// TwinCAT 3 PLC project PlcAly
// ProgramVersion: 3.1.4024.0
// libraries:
//   Tc2_EtherCAT, * (Beckhoff Automation GmbH)
//   Tc2_Standard, * (Beckhoff Automation GmbH)
//   Tc2_System, * (Beckhoff Automation GmbH)
//   Tc2_Utilities, * (Beckhoff Automation GmbH)
//   Tc3_Analytics, * (Beckhoff Automation GmbH)
//   Tc3_EventLogger, * (Beckhoff Automation GmbH)
//   Tc3_Module, * (Beckhoff Automation GmbH)
// project tree:
//   / AnalyticsTask.TcTTO, AnalyticsTask_C1.TcTTO, PlcTask.TcTTO
//   DUTs/Analytics/ E_AnalysisComponents.TcDUT, E_DataSourceContext.TcDUT, E_DataSourceState.TcDUT, E_DTType.TcDUT, E_ScopeCommand.TcDUT, E_VirtualInput.TcDUT, ST_AnalysisReset.TcDUT
//   DUTs/Analytics/HMI/Controls/ ST_HMI_C1_Ctrl1_Overall_Equipment_Effectiveness_OEE.TcDUT, ST_HMI_C1_Ctrl2_Machine_Learning_Calculation_Duration.TcDUT, ST_HMI_C1_Ctrl3_State_Unit.TcDUT
//   DUTs/Analytics/HMI/DataSourcePage/ E_SourceType.TcDUT, ST_HMI_DataSourceConfig.TcDUT, ST_HMI_DataSourceCtrl.TcDUT, ST_HMI_DataSourceHist.TcDUT, ST_HMI_DataSourceHistInfo.TcDUT, ST_HMI_DataSourceHistRecordInfo.TcDUT, ST_HMI_InputSource.TcDUT, ST_HMI_InputSourceCtrl.TcDUT
//   DUTs/Analytics/HMI/ ST_HMI_C1_OEE_Dashboard.TcDUT, ST_HMI_MapItem.TcDUT, ST_KeyValuePair.TcDUT
//   DUTs/Analytics/Sources/ ST_T1_Inputs.TcDUT
//   GVLs/ Analytics.TcGVL, AnalyticsHMI.TcGVL
//   POUs/Analytics/Analysis/ FB_Analysis.TcPOU
//   POUs/Analytics/Analysis/Networks/N01 OEEDashboard/ FB_N1_OEEDashboard.TcPOU
//   POUs/Analytics/Analysis/Networks/N01 OEEDashboard/Modules/ FB_N1_M1_State_Unit.TcPOU, FB_N1_M2_State_Execute.TcPOU, FB_N1_M3_State_Aborted.TcPOU, FB_N1_M4_State_Stopped.TcPOU, FB_N1_M5_Time_Scheduled.TcPOU, FB_N1_M6_OverallEquipmentEffectivenessOEE.TcPOU, FB_N1_M7_MachineLearningCalculationDuration.TcPOU
//   POUs/Analytics/Analysis/Networks/N01 OEEDashboard/N02 Products_Produced/ FB_N2_Products_Produced.TcPOU
//   POUs/Analytics/Analysis/Networks/N01 OEEDashboard/N02 Products_Produced/Modules/ FB_N2_M1_BatchNShift1Ch.TcPOU, FB_N2_M2_MathOperation.TcPOU, FB_N2_M3_EdgeCounter1Ch.TcPOU
//   POUs/Analytics/Analysis/Networks/N01 OEEDashboard/N03 Products_Defective/ FB_N3_Products_Defective.TcPOU
//   POUs/Analytics/Analysis/Networks/N01 OEEDashboard/N03 Products_Defective/Modules/ FB_N3_M1_BatchNShift1Ch.TcPOU, FB_N3_M2_MathOperation.TcPOU, FB_N3_M3_EdgeCounter1Ch.TcPOU
//   POUs/Analytics/Lambda/ FB_L1_Lf_CppModuleAssignString.TcPOU
//   POUs/Analytics/ MAIN_Analytics.TcPOU, MAIN_Analytics_C1.TcPOU
//   POUs/Analytics/Sources/T1_InputSource/ FB_T1_InputSource.TcPOU
//   POUs/Analytics/Sources/[Interfaces]/ I_InputSource.TcIO, I_InputSourceHistorical.TcIO
//   POUs/Analytics/VirtualInputSources/C1_AlyConfig/ FB_V1_C1_Virtual_Input_Source.TcPOU
//   POUs/Analytics/VirtualInputSources/[Interfaces]/ I_V1_Virtual_Input_Source.TcIO, I_VirtualInputSource.TcIO
//   POUs/Analytics/[Helper]/ FB_DataBuffer.TcPOU, FB_GetSampleIndex.TcPOU, FB_TcMessageSuccess.TcPOU, F_AlyTimestampToDCTimestruct.TcPOU, F_AlyTimestampToFileTime.TcPOU, F_AlyTimestampToLocalTime.TcPOU, F_ANY_Negation.TcPOU, F_ARRAY_To_LREAL_ARRAY.TcPOU, F_DCTimestructToFileTime.TcPOU, F_FileTimeToDCTimestruct.TcPOU, F_HasContext.TcPOU, F_SampleTimeCheck.TcPOU, F_ToANY.TcPOU
//   POUs/ MAIN.TcPOU
// (motion and I/O tree: see PLC project plc)
// real-time tasks:
//   TASK Task_Plc: cycle T#1ms, priority 5, ADS port 350
//   TASK Task_XPlanar_Hardware: cycle T#250us, priority 1, ADS port 351
//   TASK Task_XPlanar_Execute: cycle T#1ms, priority 3, ADS port 352
//   TASK Task_XPlanar_Prepare: cycle T#10ms, priority 10, ADS port 353
//   TASK Task_Job: cycle default, priority 7
//   TASK Task_Vision_Acquisition: cycle T#1ms, priority 4, ADS port 354
//   TASK Task_Vision_Display: cycle T#10ms, priority 12, ADS port 355
//   TASK Task_Vision_Execute: cycle T#10ms, priority 11, ADS port 356
//   TASK Task_IO: cycle T#50000us, priority 14, ADS port 301
//   TASK PlcTask: cycle T#10ms, priority 20, ADS port 357
//   TASK AnalyticsTask: cycle T#10ms, priority 21, ADS port 358
//   TASK AnalyticsTask_C1: cycle T#10ms, priority 22, ADS port 359
// variable links:

CONFIGURATION PlcAly
    RESOURCE PLC ON TwinCAT3
        TASK AnalyticsTask(INTERVAL := T#10ms, PRIORITY := 21);
        TASK AnalyticsTask_C1(INTERVAL := T#10ms, PRIORITY := 22);
        TASK PlcTask(INTERVAL := T#10ms, PRIORITY := 20);
        PROGRAM MAIN_Analytics WITH AnalyticsTask : MAIN_Analytics;
        PROGRAM MAIN_Analytics_C1 WITH AnalyticsTask_C1 : MAIN_Analytics_C1;
        PROGRAM MAIN WITH PlcTask : MAIN;
    END_RESOURCE
END_CONFIGURATION

// ---- DUTs/Analytics/E_AnalysisComponents.TcDUT
{attribute 'qualified_only'}
{attribute 'strict'}
TYPE E_AnalysisComponents : 
(
	All := -1,
	N1_OEEDashboard := 0,
	N1_M1_State_Unit := 1,
	N1_M2_State_Execute := 2,
	N1_M3_State_Aborted := 3,
	N1_M4_State_Stopped := 4,
	N1_M5_Time_Scheduled := 5,
	N1_M6_OverallEquipmentEffectivenessOEE := 6,
	N1_M7_MachineLearningCalculationDuration := 7,
	N2_Products_Produced := 8,
	N2_M1_BatchNShift1Ch := 9,
	N2_M2_MathOperation := 10,
	N2_M3_EdgeCounter1Ch := 11,
	N3_Products_Defective := 12,
	N3_M1_BatchNShift1Ch := 13,
	N3_M2_MathOperation := 14,
	N3_M3_EdgeCounter1Ch := 15,
	V1_Virtual_Input_Source := 16
) ;
END_TYPE

// ---- DUTs/Analytics/E_DataSourceContext.TcDUT
{attribute 'qualified_only'}
TYPE E_DataSourceContext : 
(
	eContext_No := 0, 
	eContext_Unknown := 2#0000_0000_0000_0001, //Unknown - All contexts allowed
	eContext_1000 := 2#0000_0000_0000_0010, //1000 µs
	eContext_Reserve1 := 2#0000_0000_0000_0100, //Reserve
	eContext_Reserve2 := 2#0000_0000_0000_1000, //Reserve
	eContext_Reserve3 := 2#0000_0000_0001_0000, //Reserve
	eContext_Reserve4 := 2#0000_0000_0010_0000, //Reserve
	eContext_Reserve5 := 2#0000_0000_0100_0000, //Reserve
	eContext_Reserve6 := 2#0000_0000_1000_0000, //Reserve
	eContext_Reserve7 := 2#0000_0001_0000_0000, //Reserve
	eContext_Reserve8 := 2#0000_0010_0000_0000, //Reserve
	eContext_Reserve9 := 2#0000_0100_0000_0000, //Reserve
	eContext_Reserve10 := 2#0000_1000_0000_0000, //Reserve
	eContext_Reserve11 := 2#0001_0000_0000_0000, //Reserve
	eContext_Reserve12 := 2#0010_0000_0000_0000, //Reserve
	eContext_Reserve13 := 2#0100_0000_0000_0000, //Reserve
	eContext_Reserve14 := 2#1000_0000_0000_0000 //Reserve
) DWORD;
END_TYPE

// ---- DUTs/Analytics/E_DataSourceState.TcDUT
{attribute 'qualified_only'}
{attribute 'strict'}
TYPE E_DataSourceState : 
(
	eUnknown := 0,
	eNotConnected,
	eReceiveData,
	eReceiveData_Cancel,
	eReceiveData_Pause,
	eError,
	eReady,
	eWaitForData
) ;
END_TYPE

// ---- DUTs/Analytics/E_DTType.TcDUT
{attribute 'qualified_only'}
{attribute 'strict'}
TYPE E_DTType : 
(
	NotInitialized := 0,
	BOOL_,
	BYTE_,
	WORD_,
	DWORD_,
	SINT_,
	USINT_,
	INT_,
	UINT_,
	DINT_,
	UDINT_,
	LINT_,
	ULINT_,
	REAL_,
	LREAL_,
	LWORD_
) ;
END_TYPE

// ---- DUTs/Analytics/E_ScopeCommand.TcDUT
{attribute 'qualified_only'}
{attribute 'strict'}
TYPE E_ScopeCommand : 
(
	eDefault := 0,
	ePause,
	eStop
) ;
END_TYPE

// ---- DUTs/Analytics/E_VirtualInput.TcDUT
{attribute 'qualified_only'}
TYPE E_VirtualInput : 
(
	eContext_No := 0, 
	eContext_V1_Virtual_Input_Source := 2#0000_0000_0000_0001_0000_0000_0000_0000, //Virtual_Input_Source
	eContext_Vn_Reserve1 := 2#0000_0000_0000_0010_0000_0000_0000_0000, //Reserve
	eContext_Vn_Reserve2 := 2#0000_0000_0000_0100_0000_0000_0000_0000, //Reserve
	eContext_Vn_Reserve3 := 2#0000_0000_0000_1000_0000_0000_0000_0000, //Reserve
	eContext_Vn_Reserve4 := 2#0000_0000_0001_0000_0000_0000_0000_0000, //Reserve
	eContext_Vn_Reserve5 := 2#0000_0000_0010_0000_0000_0000_0000_0000, //Reserve
	eContext_Vn_Reserve6 := 2#0000_0000_0100_0000_0000_0000_0000_0000, //Reserve
	eContext_Vn_Reserve7 := 2#0000_0000_1000_0000_0000_0000_0000_0000, //Reserve
	eContext_Vn_Reserve8 := 2#0000_0001_0000_0000_0000_0000_0000_0000, //Reserve
	eContext_Vn_Reserve9 := 2#0000_0010_0000_0000_0000_0000_0000_0000, //Reserve
	eContext_Vn_Reserve10 := 2#0000_0100_0000_0000_0000_0000_0000_0000, //Reserve
	eContext_Vn_Reserve11 := 2#0000_1000_0000_0000_0000_0000_0000_0000, //Reserve
	eContext_Vn_Reserve12 := 2#0001_0000_0000_0000_0000_0000_0000_0000, //Reserve
	eContext_Vn_Reserve13 := 2#0010_0000_0000_0000_0000_0000_0000_0000, //Reserve
	eContext_Vn_Reserve14 := 2#0100_0000_0000_0000_0000_0000_0000_0000, //Reserve
	eContext_Vn_Reserve15 := 2#1000_0000_0000_0000_0000_0000_0000_0000 //Reserve
) DWORD;
END_TYPE

// ---- DUTs/Analytics/HMI/Controls/ST_HMI_C1_Ctrl1_Overall_Equipment_Effectiveness_OEE.TcDUT
TYPE ST_HMI_C1_Ctrl1_Overall_Equipment_Effectiveness_OEE : 
STRUCT
	//Overall Equipment Effectiveness (OEE)
	bTrigReconfigure: BOOL;
	fM6_fOEE: LREAL; //Overall equipment effectiveness (OEE)
	fM6_fAvailability: LREAL; //Availability
	fM6_fPerformance: LREAL; //Performance
	fM6_fQuality: LREAL; //Quality
	fM6_fThresholdLevelOkWarning: LREAL; //Level Ok / Warning
	fM6_fThresholdLevelWarningAlarm: LREAL; //Level Warning / Alarm
	eM6_eOeeClass: E_ALY_Classification_3Cls; //OEE Classification
END_STRUCT
END_TYPE

// ---- DUTs/Analytics/HMI/Controls/ST_HMI_C1_Ctrl2_Machine_Learning_Calculation_Duration.TcDUT
TYPE ST_HMI_C1_Ctrl2_Machine_Learning_Calculation_Duration : 
STRUCT
	//Machine Learning Calculation Duration
	bTrigReconfigure: BOOL;
	nM7_nDataIn: UDINT; //Actual Value
	fM7_fMin: LREAL; //Min Value
	fM7_fMax: LREAL; //Max Value
	fM7_fAvg: LREAL; //Avg Value
	tM7_fbTimeMin: DCTIMESTRUCT; //Last Event Min
	tM7_fbTimeMax: DCTIMESTRUCT; //Last Event Max
END_STRUCT
END_TYPE

// ---- DUTs/Analytics/HMI/Controls/ST_HMI_C1_Ctrl3_State_Unit.TcDUT
TYPE ST_HMI_C1_Ctrl3_State_Unit : 
STRUCT
	//State_Unit
	bTrigReconfigure: BOOL;
	sM1_sOutput: STRING(255); //Value
END_STRUCT
END_TYPE

// ---- DUTs/Analytics/HMI/DataSourcePage/E_SourceType.TcDUT
{attribute 'qualified_only'}
{attribute 'strict'}
TYPE E_SourceType : 
(
	eLive := 0,
	eHistMQTT,
	eHistFile
) ;
END_TYPE

// ---- DUTs/Analytics/HMI/DataSourcePage/ST_HMI_DataSourceConfig.TcDUT
TYPE ST_HMI_DataSourceConfig : 
STRUCT
	nID: DINT;
	sDisplayName: WSTRING(80);
	eConfigType: E_SourceType;
	aInputSources: ARRAY [0..0] OF ST_HMI_InputSource;
END_STRUCT
END_TYPE

// ---- DUTs/Analytics/HMI/DataSourcePage/ST_HMI_DataSourceCtrl.TcDUT
TYPE ST_HMI_DataSourceCtrl : 
STRUCT
	nActiveConfigurationIdx: INT;
	
	aInputSourceCtrls: ARRAY [0..0] OF ST_HMI_InputSourceCtrl;
	
	bStart: BOOL;
	bCancel: BOOL;
	bPause: BOOL;
	bReset: BOOL;
	
	bUpdateRecordList: BOOL;
END_STRUCT
END_TYPE

// ---- DUTs/Analytics/HMI/DataSourcePage/ST_HMI_DataSourceHist.TcDUT
TYPE ST_HMI_DataSourceHist : 
STRUCT
	nCurrentRecordID: DINT;
	stSourceInfo: ST_HMI_DataSourceHistInfo;
	nRecordCount: DINT;
	aRecords: ARRAY [0..255] OF ST_HMI_DataSourceHistRecordInfo;
END_STRUCT
END_TYPE

// ---- DUTs/Analytics/HMI/DataSourcePage/ST_HMI_DataSourceHistInfo.TcDUT
TYPE ST_HMI_DataSourceHistInfo : 
STRUCT
	sSPGuid: GUID;
	sAlyFilePath: STRING(255);
	sSourceType: STRING(80);
	sTopic: STRING(255);
	sLayoutID: GUID;
	sAlias: STRING(255);
END_STRUCT
END_TYPE

// ---- DUTs/Analytics/HMI/DataSourcePage/ST_HMI_DataSourceHistRecordInfo.TcDUT
TYPE ST_HMI_DataSourceHistRecordInfo : 
STRUCT
	nID: DINT;
	sName: WSTRING(80);
	sDisplayName: WSTRING(80);
	dtRecordStart: DCTIMESTRUCT;
	dtRecordEnd: DCTIMESTRUCT;
	dtSelectedRangeStart: DCTIMESTRUCT;
	dtSelectedRangeEnd: DCTIMESTRUCT;
END_STRUCT
END_TYPE

// ---- DUTs/Analytics/HMI/DataSourcePage/ST_HMI_InputSource.TcDUT
TYPE ST_HMI_InputSource : 
STRUCT
	nID: DINT;
	sDisplayName: WSTRING(80);
	
	sStreamSystemID: GUID;
	sTopic: STRING(255);
	
	eSourceType: E_SourceType;;
	eState: E_DataSourceState;;
	dtTimestamp: DCTIMESTRUCT;
	
	stHist: ST_HMI_DataSourceHist;
END_STRUCT
END_TYPE

// ---- DUTs/Analytics/HMI/DataSourcePage/ST_HMI_InputSourceCtrl.TcDUT
TYPE ST_HMI_InputSourceCtrl : 
STRUCT
	nActiveRecordIdx: INT;
	
	dtSelectedRangeStart: DCTIMESTRUCT;
	dtSelectedRangeEnd: DCTIMESTRUCT;
	
	bStart: BOOL;
	bCancel: BOOL;
	bPause: BOOL;
	bReset: BOOL;
END_STRUCT
END_TYPE

// ---- DUTs/Analytics/HMI/ST_HMI_C1_OEE_Dashboard.TcDUT
TYPE ST_HMI_C1_OEE_Dashboard : 
STRUCT
	stHMI_C1_Ctrl3_State_Unit: ST_HMI_C1_Ctrl3_State_Unit;
	
	stHMI_C1_Ctrl1_Overall_Equipment_Effectiveness_OEE: ST_HMI_C1_Ctrl1_Overall_Equipment_Effectiveness_OEE;
	
	stHMI_C1_Ctrl2_Machine_Learning_Calculation_Duration: ST_HMI_C1_Ctrl2_Machine_Learning_Calculation_Duration;
END_STRUCT
END_TYPE

// ---- DUTs/Analytics/HMI/ST_HMI_MapItem.TcDUT
TYPE ST_HMI_MapItem : 
STRUCT
	sName: WSTRING(127);
	sDescription: WSTRING(127);
	sPosition: WSTRING(127);
	nStatus: INT;
END_STRUCT
END_TYPE

// ---- DUTs/Analytics/HMI/ST_KeyValuePair.TcDUT
TYPE ST_KeyValuePair : 
STRUCT
	sKey: WSTRING(127);
	sValue: STRING(255);
END_STRUCT
END_TYPE

// ---- DUTs/Analytics/Sources/ST_T1_Inputs.TcDUT
TYPE ST_T1_Inputs : 
STRUCT
	nGVL_Components_fbMachine_stAnalytics_nState: UINT; //GVL_Components.fbMachine.stAnalytics.nState
	nGVL_Components_fbMachine_stAnalytics_nUnitsProduced: ULINT; //GVL_Components.fbMachine.stAnalytics.nUnitsProduced
	nGVL_Components_fbMachine_stAnalytics_nDefectiveUnits: ULINT; //GVL_Components.fbMachine.stAnalytics.nDefectiveUnits
	nGVL_Components_fbMachine_stAnalytics_tMlCalculation: UDINT; //GVL_Components.fbMachine.stAnalytics.tMlCalculation
END_STRUCT
END_TYPE

// ---- DUTs/Analytics/ST_AnalysisReset.TcDUT
TYPE ST_AnalysisReset : 
STRUCT
	eResetComponent: E_AnalysisComponents := E_AnalysisComponents.All;
	bResetExecute: BOOL;
END_STRUCT
END_TYPE

// ---- GVLs/Analytics.TcGVL
{attribute 'qualified_only'}
VAR_GLOBAL
	//DataSources
	//Live:
	fbT1_InputSource: FB_T1_InputSource;
	//Historical:
	//Empty:
	
	fbT1_IecCriticalSection: FB_IecCriticalSection;
	
	//Historical DataSource parameter
	nHistMaxInputBuffer: UDINT := 100;
	nHistMaxSampleCount: UDINT := 100;
	
	stReset: ST_AnalysisReset;
END_VAR

// ---- GVLs/AnalyticsHMI.TcGVL
{attribute 'qualified_only'}
VAR_GLOBAL
	//Switch between historical and live data
	stHMI_DataSourceCtrl: ST_HMI_DataSourceCtrl;
	stHMI_DataSourceConfig: ARRAY [0..0] OF ST_HMI_DataSourceConfig := [ 
																	( nID:= 1, sDisplayName:= "AlyConfig", eConfigType:= E_SourceType.eLive, 
																		aInputSources:= [ 
																			( nID:= 1, sDisplayName:= "00436273-58a1-a0ec-e33c-07029f4f38f0", sStreamSystemID:= STRING_TO_GUID('00436273-58a1-a0ec-e33c-07029f4f38f0'), 
																				sTopic:= 'DefaultMainTopic/PlcStream1', eSourceType:= E_SourceType.eLive, eState:= E_DataSourceState.eUnknown ) ] ) ];
	
	//Reset
	bN1_OEEDashboard_Reset: BOOL;
	bN1_M1_State_Unit_Reset: BOOL;
	bN1_M2_State_Execute_Reset: BOOL;
	bN1_M3_State_Aborted_Reset: BOOL;
	bN1_M4_State_Stopped_Reset: BOOL;
	bN1_M5_Time_Scheduled_Reset: BOOL;
	bN1_M6_OverallEquipmentEffectivenessOEE_Reset: BOOL;
	bN1_M7_MachineLearningCalculationDuration_Reset: BOOL;
	bN2_Products_Produced_Reset: BOOL;
	bN2_M1_BatchNShift1Ch_Reset: BOOL;
	bN2_M2_MathOperation_Reset: BOOL;
	bN2_M3_EdgeCounter1Ch_Reset: BOOL;
	bN3_Products_Defective_Reset: BOOL;
	bN3_M1_BatchNShift1Ch_Reset: BOOL;
	bN3_M2_MathOperation_Reset: BOOL;
	bN3_M3_EdgeCounter1Ch_Reset: BOOL;
	
	//HMI Structs
	stHMI_C1_OEE_Dashboard: ST_HMI_C1_OEE_Dashboard;
	
	//HMI Map Items
	aMapItems: ARRAY [0..0] OF ST_HMI_MapItem := [(sName:="00436273-58a1-a0ec-e33c-07029f4f38f0", sDescription:="", sPosition:="", nStatus:= 0)];
END_VAR

// ---- POUs/Analytics/Sources/[Interfaces]/I_InputSource.TcIO
INTERFACE I_InputSource

METHOD AddClient : BOOL
VAR_OUTPUT
	nClientID: LWORD;
END_VAR
END_METHOD

METHOD Call : BOOL
END_METHOD

METHOD ClientDone : BOOL
VAR_INPUT
	nClientID: LWORD;
END_VAR
END_METHOD

METHOD GetData : BOOL
VAR_INPUT
	nElement: UDINT;
	pInputs: PVOID;
	nInputsSize: UDINT;
END_VAR
VAR_OUTPUT
	nTimestamp: ULINT;
	nContext: DWORD;
END_VAR
END_METHOD

METHOD NewDataAvailable : BOOL
VAR_INPUT
	nLastDataHandle: ULINT;
END_VAR
END_METHOD

PROPERTY eDataState : E_DataSourceState
GET
END_GET
END_PROPERTY

PROPERTY bReadNewData : BOOL
GET
END_GET
END_PROPERTY

PROPERTY nDataHandle : ULINT
GET
END_GET
END_PROPERTY

PROPERTY nElements : UDINT
GET
END_GET
END_PROPERTY

PROPERTY nMaxOversamplingFactor : UDINT
GET
END_GET
END_PROPERTY

END_INTERFACE

// ---- POUs/Analytics/Sources/[Interfaces]/I_InputSourceHistorical.TcIO
INTERFACE I_InputSourceHistorical EXTENDS I_InputSource

METHOD HistoricalCtrl : BOOL
VAR_INPUT
	stCtrl: REFERENCE TO ST_HMI_InputSourceCtrl;
	stHistStreamInfo: REFERENCE TO ST_HMI_DataSourceHist;
	stRecordInfo: REFERENCE TO ST_HMI_DataSourceHistRecordInfo;
END_VAR
END_METHOD

METHOD UpdateRecordList : BOOL
VAR_INPUT
	sStreamSystemID: GUID;
	stHistStreamInfo: REFERENCE TO ST_HMI_DataSourceHist;
END_VAR
END_METHOD

PROPERTY bCtrlChanged : BOOL
GET
END_GET
END_PROPERTY

END_INTERFACE

// ---- POUs/Analytics/VirtualInputSources/[Interfaces]/I_V1_Virtual_Input_Source.TcIO
INTERFACE I_V1_Virtual_Input_Source EXTENDS I_VirtualInputSource

PROPERTY nV1_tMlCalculation : UDINT
GET
END_GET
END_PROPERTY

PROPERTY nV1_nUnitsProduced : ULINT
GET
END_GET
END_PROPERTY

PROPERTY nV1_nDefectiveUnits : ULINT
GET
END_GET
END_PROPERTY

PROPERTY nV1_nState : UINT
GET
END_GET
END_PROPERTY

END_INTERFACE

// ---- POUs/Analytics/VirtualInputSources/[Interfaces]/I_VirtualInputSource.TcIO
INTERFACE I_VirtualInputSource

METHOD Done : BOOL
END_METHOD

METHOD NextData : BOOL
VAR_INPUT
	nMaxOversampling: UDINT;
END_VAR
END_METHOD

METHOD SourceSync : BOOL
END_METHOD

PROPERTY bEndOfData : BOOL
GET
END_GET
END_PROPERTY

PROPERTY dtTimestamp : DCTIMESTRUCT
GET
END_GET
END_PROPERTY

PROPERTY nContext : DWORD
GET
END_GET
END_PROPERTY

PROPERTY nDataHandle : ULINT
GET
END_GET
END_PROPERTY

PROPERTY tTimestamp : ULINT
GET
END_GET
END_PROPERTY

PROPERTY eSourceState : E_DataSourceState
GET
END_GET
END_PROPERTY

END_INTERFACE

// ---- POUs/Analytics/MAIN_Analytics.TcPOU
PROGRAM MAIN_Analytics
VAR
END_VAR


//Reset Analytics Components
A_Reset();

CASE AnalyticsHMI.stHMI_DataSourceCtrl.nActiveConfigurationIdx OF
	0:

		//Reset
		MAIN_Analytics_C1.A_Reset(stReset := Analytics.stReset);

		//Map to HMI
		MAIN_Analytics_C1.A_MapToHMI();
END_CASE


//Call DataSource FBs
IF Analytics.fbT1_InputSource.bReadNewData THEN
	Analytics.fbT1_InputSource.Call();
END_IF

ACTION A_Reset:

IF AnalyticsHMI.bN1_OEEDashboard_Reset THEN
	Analytics.stReset.eResetComponent:= E_AnalysisComponents.N1_OEEDashboard;
	Analytics.stReset.bResetExecute:= TRUE;
	AnalyticsHMI.bN1_OEEDashboard_Reset:= FALSE;
END_IF

IF AnalyticsHMI.bN1_M1_State_Unit_Reset THEN
	Analytics.stReset.eResetComponent:= E_AnalysisComponents.N1_M1_State_Unit;
	Analytics.stReset.bResetExecute:= TRUE;
	AnalyticsHMI.bN1_M1_State_Unit_Reset:= FALSE;
END_IF

IF AnalyticsHMI.bN1_M2_State_Execute_Reset THEN
	Analytics.stReset.eResetComponent:= E_AnalysisComponents.N1_M2_State_Execute;
	Analytics.stReset.bResetExecute:= TRUE;
	AnalyticsHMI.bN1_M2_State_Execute_Reset:= FALSE;
END_IF

IF AnalyticsHMI.bN1_M3_State_Aborted_Reset THEN
	Analytics.stReset.eResetComponent:= E_AnalysisComponents.N1_M3_State_Aborted;
	Analytics.stReset.bResetExecute:= TRUE;
	AnalyticsHMI.bN1_M3_State_Aborted_Reset:= FALSE;
END_IF

IF AnalyticsHMI.bN1_M4_State_Stopped_Reset THEN
	Analytics.stReset.eResetComponent:= E_AnalysisComponents.N1_M4_State_Stopped;
	Analytics.stReset.bResetExecute:= TRUE;
	AnalyticsHMI.bN1_M4_State_Stopped_Reset:= FALSE;
END_IF

IF AnalyticsHMI.bN1_M5_Time_Scheduled_Reset THEN
	Analytics.stReset.eResetComponent:= E_AnalysisComponents.N1_M5_Time_Scheduled;
	Analytics.stReset.bResetExecute:= TRUE;
	AnalyticsHMI.bN1_M5_Time_Scheduled_Reset:= FALSE;
END_IF

IF AnalyticsHMI.bN1_M6_OverallEquipmentEffectivenessOEE_Reset THEN
	Analytics.stReset.eResetComponent:= E_AnalysisComponents.N1_M6_OverallEquipmentEffectivenessOEE;
	Analytics.stReset.bResetExecute:= TRUE;
	AnalyticsHMI.bN1_M6_OverallEquipmentEffectivenessOEE_Reset:= FALSE;
END_IF

IF AnalyticsHMI.bN1_M7_MachineLearningCalculationDuration_Reset THEN
	Analytics.stReset.eResetComponent:= E_AnalysisComponents.N1_M7_MachineLearningCalculationDuration;
	Analytics.stReset.bResetExecute:= TRUE;
	AnalyticsHMI.bN1_M7_MachineLearningCalculationDuration_Reset:= FALSE;
END_IF

IF AnalyticsHMI.bN2_Products_Produced_Reset THEN
	Analytics.stReset.eResetComponent:= E_AnalysisComponents.N2_Products_Produced;
	Analytics.stReset.bResetExecute:= TRUE;
	AnalyticsHMI.bN2_Products_Produced_Reset:= FALSE;
END_IF

IF AnalyticsHMI.bN2_M1_BatchNShift1Ch_Reset THEN
	Analytics.stReset.eResetComponent:= E_AnalysisComponents.N2_M1_BatchNShift1Ch;
	Analytics.stReset.bResetExecute:= TRUE;
	AnalyticsHMI.bN2_M1_BatchNShift1Ch_Reset:= FALSE;
END_IF

IF AnalyticsHMI.bN2_M2_MathOperation_Reset THEN
	Analytics.stReset.eResetComponent:= E_AnalysisComponents.N2_M2_MathOperation;
	Analytics.stReset.bResetExecute:= TRUE;
	AnalyticsHMI.bN2_M2_MathOperation_Reset:= FALSE;
END_IF

IF AnalyticsHMI.bN2_M3_EdgeCounter1Ch_Reset THEN
	Analytics.stReset.eResetComponent:= E_AnalysisComponents.N2_M3_EdgeCounter1Ch;
	Analytics.stReset.bResetExecute:= TRUE;
	AnalyticsHMI.bN2_M3_EdgeCounter1Ch_Reset:= FALSE;
END_IF

IF AnalyticsHMI.bN3_Products_Defective_Reset THEN
	Analytics.stReset.eResetComponent:= E_AnalysisComponents.N3_Products_Defective;
	Analytics.stReset.bResetExecute:= TRUE;
	AnalyticsHMI.bN3_Products_Defective_Reset:= FALSE;
END_IF

IF AnalyticsHMI.bN3_M1_BatchNShift1Ch_Reset THEN
	Analytics.stReset.eResetComponent:= E_AnalysisComponents.N3_M1_BatchNShift1Ch;
	Analytics.stReset.bResetExecute:= TRUE;
	AnalyticsHMI.bN3_M1_BatchNShift1Ch_Reset:= FALSE;
END_IF

IF AnalyticsHMI.bN3_M2_MathOperation_Reset THEN
	Analytics.stReset.eResetComponent:= E_AnalysisComponents.N3_M2_MathOperation;
	Analytics.stReset.bResetExecute:= TRUE;
	AnalyticsHMI.bN3_M2_MathOperation_Reset:= FALSE;
END_IF

IF AnalyticsHMI.bN3_M3_EdgeCounter1Ch_Reset THEN
	Analytics.stReset.eResetComponent:= E_AnalysisComponents.N3_M3_EdgeCounter1Ch;
	Analytics.stReset.bResetExecute:= TRUE;
	AnalyticsHMI.bN3_M3_EdgeCounter1Ch_Reset:= FALSE;
END_IF
END_ACTION

END_PROGRAM

// ---- POUs/Analytics/MAIN_Analytics_C1.TcPOU
PROGRAM MAIN_Analytics_C1
VAR_INPUT
	stReset: ST_AnalysisReset;
END_VAR
VAR_OUTPUT
	bError: BOOL;
	ipTcResult: I_TcMessage;
END_VAR
VAR
	nHMIUpdateState: INT;
	bHMIReinit: BOOL := TRUE;
	bHMIResetReinit: BOOL;
	bHMIReinitDone: BOOL;
	
	fbV1_C1_Virtual_Input_Source: FB_V1_C1_Virtual_Input_Source(fbSource:= Analytics.fbT1_InputSource);
	
	fbAnalysis: FB_Analysis := ( nConfigurationID:= 1, 
								ipVirtual_Input_Source:= fbV1_C1_Virtual_Input_Source );
END_VAR

A_Reset();

fbV1_C1_Virtual_Input_Source.SourceSync();

IF NOT fbV1_C1_Virtual_Input_Source.bEndOfData THEN

	WHILE NOT fbV1_C1_Virtual_Input_Source.bEndOfData DO

		fbV1_C1_Virtual_Input_Source.NextData(1);

		fbAnalysis.Call();

	END_WHILE

ELSE
	fbAnalysis.Call();
END_IF

fbV1_C1_Virtual_Input_Source.Done();

//Error Handling
bError:= fbAnalysis.bError;
ipTcResult:= fbAnalysis.ipTcResult;


//Map HMI Current Timestamp
AnalyticsHMI.stHMI_DataSourceConfig[0].aInputSources[0].eState:= fbV1_C1_Virtual_Input_Source.fbInputSource.eDataState;
AnalyticsHMI.stHMI_DataSourceConfig[0].aInputSources[0].dtTimestamp:= fbV1_C1_Virtual_Input_Source.dtTimestamp;

ACTION A_Reset:

//Reset Analytics Components
fbAnalysis.Reset(stReset);

Analytics.stReset.bResetExecute:= FALSE;
END_ACTION

ACTION A_MapToHMI:

//Map In-/Outputs of the Analysis to HMI Structs
CASE nHMIUpdateState OF
	0:
		bHMIReinit:= bHMIReinit OR fbAnalysis.GetHMIValues(1, ADR(AnalyticsHMI.stHMI_C1_OEE_Dashboard));
		bHMIReinitDone:= fbAnalysis.SetHMIValues(1, ADR(AnalyticsHMI.stHMI_C1_OEE_Dashboard), bHMIReinit);
		nHMIUpdateState:= 1;
	1:
		IF bHMIResetReinit THEN
			bHMIResetReinit:= FALSE;
			bHMIReinit:= FALSE;
		END_IF

		IF bHMIReinitDone THEN
			bHMIResetReinit:= TRUE;
		END_IF

		nHMIUpdateState:= 0;
END_CASE
END_ACTION

END_PROGRAM

// ---- POUs/Analytics/VirtualInputSources/C1_AlyConfig/FB_V1_C1_Virtual_Input_Source.TcPOU
FUNCTION_BLOCK FB_V1_C1_Virtual_Input_Source IMPLEMENTS I_VirtualInputSource, I_V1_Virtual_Input_Source
VAR
	_fbSource: I_InputSource;
	
	_nSourceClientID: LWORD;
	_nDataHandle: ULINT;
	_nElements: UDINT;
	
	_nSelectedElement: UDINT;
	_nSelectedOversample: UDINT;
	
	_nContext: DWORD;
	_stInputs: ST_T1_Inputs;
	
	_nTimestamp: ULINT;
END_VAR

PROPERTY bEndOfData : BOOL
GET
bEndOfData:= _nElements = 0 OR (_nSelectedElement >= _nElements AND _nSelectedOversample >= _fbSource.nMaxOversamplingFactor);
END_GET
END_PROPERTY

METHOD Done : BOOL
VAR
END_VAR
IF bEndOfData AND _nElements > 0 THEN
	_nElements:= 0;
	_fbSource.ClientDone(_nSourceClientID);
END_IF

_nContext:= 0;
END_METHOD

PROPERTY dtTimestamp : DCTIMESTRUCT
GET
dtTimestamp:= F_AlyTimestampToDCTimestruct(_nTimestamp);
END_GET
END_PROPERTY

PROPERTY eSourceState : E_DataSourceState
GET
eSourceState:= _fbSource.eDataState;
END_GET
END_PROPERTY

METHOD FB_init : BOOL
VAR_INPUT
	bInitRetains: BOOL; // if TRUE, the retain variables are initialized (warm start / cold start)
	bInCopyCode: BOOL; // if TRUE, the instance afterwards gets moved into the copy code (online change)
	fbSource: I_InputSource;
END_VAR
VAR
END_VAR
IF NOT bInCopyCode THEN
	fbSource.AddClient(nClientID=>_nSourceClientID);
	_fbSource:= fbSource;
END_IF
END_METHOD

PROPERTY fbInputSource : I_InputSource
GET
fbInputSource:= _fbSource;
END_GET
END_PROPERTY

PROPERTY nContext : DWORD
GET
nContext:= _nContext;
END_GET
END_PROPERTY

PROPERTY nDataHandle : ULINT
GET
nDataHandle:= _nDataHandle;
END_GET
END_PROPERTY

METHOD NextData : BOOL
VAR_INPUT
	nMaxOversampling: UDINT;
END_VAR
VAR
END_VAR
IF _nElements > 0 AND NOT bEndOfData THEN

	_nSelectedOversample:= _nSelectedOversample + 1;
	IF _nSelectedOversample > nMaxOversampling OR _nSelectedElement = 0 THEN
		_nSelectedElement:= _nSelectedElement + 1;
		_nSelectedOversample:= 1;
	END_IF

	NextData:= _fbSource.GetData(_nSelectedElement, ADR(_stInputs), SIZEOF(_stInputs), nTimestamp=>_nTimestamp, nContext=>_nContext);
	_nContext:= _nContext OR E_VirtualInput.eContext_V1_Virtual_Input_Source;
END_IF
END_METHOD

PROPERTY nV1_nDefectiveUnits : ULINT
GET
nV1_nDefectiveUnits:= _stInputs.nGVL_Components_fbMachine_stAnalytics_nDefectiveUnits;
END_GET
END_PROPERTY

PROPERTY nV1_nState : UINT
GET
nV1_nState:= _stInputs.nGVL_Components_fbMachine_stAnalytics_nState;
END_GET
END_PROPERTY

PROPERTY nV1_nUnitsProduced : ULINT
GET
nV1_nUnitsProduced:= _stInputs.nGVL_Components_fbMachine_stAnalytics_nUnitsProduced;
END_GET
END_PROPERTY

PROPERTY nV1_tMlCalculation : UDINT
GET
nV1_tMlCalculation:= _stInputs.nGVL_Components_fbMachine_stAnalytics_tMlCalculation;
END_GET
END_PROPERTY

METHOD SourceSync : BOOL
VAR
END_VAR
IF _fbSource.NewDataAvailable(_nDataHandle) THEN
	_nDataHandle:= _fbSource.nDataHandle;
	_nElements:= _fbSource.nElements;

	_nSelectedElement:= 0;
	_nSelectedOversample:= 0;
END_IF
END_METHOD

PROPERTY tTimestamp : ULINT
GET
tTimestamp:= _nTimestamp;
END_GET
END_PROPERTY

END_FUNCTION_BLOCK

// ---- POUs/Analytics/[Helper]/F_AlyTimestampToDCTimestruct.TcPOU
FUNCTION F_AlyTimestampToDCTimestruct : DCTIMESTRUCT
VAR_INPUT
	tTimestamp: ULINT;
END_VAR
VAR
	tFileTime: T_FILETIME;
	newDCTime: T_DCTIME64;
	
	fbToLocal: FB_FileTimeToTzSpecificLocalTime;
	//W. Europe Daylight Time
	//(UTC+01:00) Amsterdam, Berlin, Bern, Rome, Stockholm, Vienna
	tzInfo: ST_TimeZoneInformation := (bias := -60, standardDate := (wMonth := 10 ,wDay:=5, wHour := 3), daylightDate := (wMonth := 3, wDay:=5, wHour := 2), daylightBias := -60);
END_VAR

tFileTime:= DCTIME64_TO_Filetime(tTimestamp);
fbToLocal(in:= tFileTime, tzInfo:= tzInfo);
newDCTime:= FILETIME_TO_DCTIME64(fbToLocal.out);

F_AlyTimestampToDCTimestruct:= DCTIME64_TO_DCTIMESTRUCT(newDCTime);

END_FUNCTION

// ---- POUs/Analytics/Analysis/FB_Analysis.TcPOU
FUNCTION_BLOCK FB_Analysis
VAR_INPUT
	nConfigurationID: INT;
	ipVirtual_Input_Source: I_V1_Virtual_Input_Source;
	
END_VAR
VAR_OUTPUT
	bError: BOOL;
	ipTcResult: I_TcMessage := fbTcMsgSuccess;
END_VAR
VAR
	fbTcMsgSuccess: FB_TcMessageSuccess;
	
	R_TRIG_Reset: R_TRIG;
	bResetBusy: BOOL;
	
	fbN1_OEEDashboard: FB_N1_OEEDashboard;
END_VAR

METHOD Call : BOOL
VAR
END_VAR

//Analytics Network "OEEDashboard" with ID: 1
fbN1_OEEDashboard.Call(THIS);


//Error Handling
IF fbN1_OEEDashboard.bError THEN
	bError:= TRUE;
	ipTcResult:= fbN1_OEEDashboard.ipTcResult;
ELSE
	bError:= FALSE;
	ipTcResult:= fbTcMsgSuccess;
END_IF
END_METHOD

METHOD GetHMIValues : BOOL
VAR_INPUT
	nContentID: DINT;
	pContent: PVOID;
END_VAR
VAR
END_VAR

CASE nContentID OF
	1:
		GetHMIValues:= GetHMIValues OR fbN1_OEEDashboard.fbM6_OverallEquipmentEffectivenessOEE.GetHMI(1, pContent);
END_CASE
END_METHOD

PROPERTY nContext : DWORD
GET

nContext:= 0;
IF ipVirtual_Input_Source <> 0 THEN
	nContext:= ipVirtual_Input_Source.nContext;
END_IF
END_GET
END_PROPERTY

METHOD Reset : BOOL
VAR_IN_OUT
	stReset: ST_AnalysisReset;
END_VAR
VAR
END_VAR

R_TRIG_Reset(CLK:= stReset.bResetExecute);
IF R_TRIG_Reset.Q OR bResetBusy THEN
	bResetBusy:= TRUE;

	CASE stReset.eResetComponent OF
		E_AnalysisComponents.All:
			bResetBusy:= bResetBusy AND fbN1_OEEDashboard.Reset();
			bResetBusy:= bResetBusy AND fbN1_OEEDashboard.fbN2_Products_Produced.Reset();
			bResetBusy:= bResetBusy AND fbN1_OEEDashboard.fbN3_Products_Defective.Reset();
		E_AnalysisComponents.N1_OEEDashboard:
			bResetBusy:= bResetBusy AND fbN1_OEEDashboard.Reset();
		E_AnalysisComponents.N1_M1_State_Unit:
			bResetBusy:= bResetBusy AND fbN1_OEEDashboard.fbM1_State_Unit.Reset();
		E_AnalysisComponents.N1_M2_State_Execute:
			bResetBusy:= bResetBusy AND fbN1_OEEDashboard.fbM2_State_Execute.Reset();
		E_AnalysisComponents.N1_M3_State_Aborted:
			bResetBusy:= bResetBusy AND fbN1_OEEDashboard.fbM3_State_Aborted.Reset();
		E_AnalysisComponents.N1_M4_State_Stopped:
			bResetBusy:= bResetBusy AND fbN1_OEEDashboard.fbM4_State_Stopped.Reset();
		E_AnalysisComponents.N1_M5_Time_Scheduled:
			bResetBusy:= bResetBusy AND fbN1_OEEDashboard.fbM5_Time_Scheduled.Reset();
		E_AnalysisComponents.N1_M6_OverallEquipmentEffectivenessOEE:
			bResetBusy:= bResetBusy AND fbN1_OEEDashboard.fbM6_OverallEquipmentEffectivenessOEE.Reset();
		E_AnalysisComponents.N1_M7_MachineLearningCalculationDuration:
			bResetBusy:= bResetBusy AND fbN1_OEEDashboard.fbM7_MachineLearningCalculationDuration.Reset();
		E_AnalysisComponents.N2_Products_Produced:
			bResetBusy:= bResetBusy AND fbN1_OEEDashboard.fbN2_Products_Produced.Reset();
		E_AnalysisComponents.N2_M1_BatchNShift1Ch:
			bResetBusy:= bResetBusy AND fbN1_OEEDashboard.fbN2_Products_Produced.fbM1_BatchNShift1Ch.Reset();
		E_AnalysisComponents.N2_M2_MathOperation:
			bResetBusy:= bResetBusy AND fbN1_OEEDashboard.fbN2_Products_Produced.fbM2_MathOperation.Reset();
		E_AnalysisComponents.N2_M3_EdgeCounter1Ch:
			bResetBusy:= bResetBusy AND fbN1_OEEDashboard.fbN2_Products_Produced.fbM3_EdgeCounter1Ch.Reset();
		E_AnalysisComponents.N3_Products_Defective:
			bResetBusy:= bResetBusy AND fbN1_OEEDashboard.fbN3_Products_Defective.Reset();
		E_AnalysisComponents.N3_M1_BatchNShift1Ch:
			bResetBusy:= bResetBusy AND fbN1_OEEDashboard.fbN3_Products_Defective.fbM1_BatchNShift1Ch.Reset();
		E_AnalysisComponents.N3_M2_MathOperation:
			bResetBusy:= bResetBusy AND fbN1_OEEDashboard.fbN3_Products_Defective.fbM2_MathOperation.Reset();
		E_AnalysisComponents.N3_M3_EdgeCounter1Ch:
			bResetBusy:= bResetBusy AND fbN1_OEEDashboard.fbN3_Products_Defective.fbM3_EdgeCounter1Ch.Reset();
		E_AnalysisComponents.V1_Virtual_Input_Source:
			bResetBusy:= bResetBusy AND fbN1_OEEDashboard.fbM1_State_Unit.Reset();
			bResetBusy:= bResetBusy AND fbN1_OEEDashboard.fbM2_State_Execute.Reset();
			bResetBusy:= bResetBusy AND fbN1_OEEDashboard.fbM3_State_Aborted.Reset();
			bResetBusy:= bResetBusy AND fbN1_OEEDashboard.fbM4_State_Stopped.Reset();
			bResetBusy:= bResetBusy AND fbN1_OEEDashboard.fbM5_Time_Scheduled.Reset();
			bResetBusy:= bResetBusy AND fbN1_OEEDashboard.fbM6_OverallEquipmentEffectivenessOEE.Reset();
			bResetBusy:= bResetBusy AND fbN1_OEEDashboard.fbM7_MachineLearningCalculationDuration.Reset();
			bResetBusy:= bResetBusy AND fbN1_OEEDashboard.fbN2_Products_Produced.fbM1_BatchNShift1Ch.Reset();
			bResetBusy:= bResetBusy AND fbN1_OEEDashboard.fbN2_Products_Produced.fbM2_MathOperation.Reset();
			bResetBusy:= bResetBusy AND fbN1_OEEDashboard.fbN2_Products_Produced.fbM3_EdgeCounter1Ch.Reset();
			bResetBusy:= bResetBusy AND fbN1_OEEDashboard.fbN3_Products_Defective.fbM1_BatchNShift1Ch.Reset();
			bResetBusy:= bResetBusy AND fbN1_OEEDashboard.fbN3_Products_Defective.fbM2_MathOperation.Reset();
			bResetBusy:= bResetBusy AND fbN1_OEEDashboard.fbN3_Products_Defective.fbM3_EdgeCounter1Ch.Reset();
	END_CASE

	bResetBusy:= NOT bResetBusy;

	stReset.bResetExecute:= bResetBusy;
END_IF
END_METHOD

METHOD SetHMIValues : BOOL
VAR_INPUT
	nContentID: DINT;
	pContent: PVOID;
	bHMIReinit: BOOL;
END_VAR
VAR
END_VAR

CASE nContentID OF
	1:
		SetHMIValues:= fbN1_OEEDashboard.fbM1_State_Unit.SetHMI(1, pContent, bHMIReinit);
		SetHMIValues:= SetHMIValues AND fbN1_OEEDashboard.fbM6_OverallEquipmentEffectivenessOEE.SetHMI(1, pContent, bHMIReinit);
		SetHMIValues:= SetHMIValues AND fbN1_OEEDashboard.fbM7_MachineLearningCalculationDuration.SetHMI(1, pContent, bHMIReinit);
END_CASE
END_METHOD

END_FUNCTION_BLOCK

// ---- POUs/Analytics/[Helper]/FB_TcMessageSuccess.TcPOU
FUNCTION_BLOCK FB_TcMessageSuccess EXTENDS FB_TcMessage
VAR
END_VAR

METHOD FB_init : BOOL
VAR_INPUT
	bInitRetains: BOOL; // if TRUE, the retain variables are initialized (warm start / cold start)
	bInCopyCode: BOOL; // if TRUE, the instance afterwards gets moved into the copy code (online change)
END_VAR
VAR
END_VAR
IF NOT bInCopyCode THEN
	SUPER^.CreateEx(Tc3_EventLogger.SUCCESS_EVENT, 0);
END_IF
END_METHOD

END_FUNCTION_BLOCK

// ---- POUs/Analytics/Analysis/Networks/N01 OEEDashboard/FB_N1_OEEDashboard.TcPOU
//Analytics Network "OEEDashboard" with ID: 1
{attribute 'no_assign'}
FUNCTION_BLOCK FB_N1_OEEDashboard
VAR_OUTPUT
	bError: BOOL;
	ipTcResult: I_TcMessage := fbTcMsgSuccess;
END_VAR
VAR
	fbTcMsgSuccess: FB_TcMessageSuccess;
	
	//Modules
	fbM1_State_Unit: FB_N1_M1_State_Unit;
	fbM2_State_Execute: FB_N1_M2_State_Execute;
	fbM3_State_Aborted: FB_N1_M3_State_Aborted;
	fbM4_State_Stopped: FB_N1_M4_State_Stopped;
	fbM5_Time_Scheduled: FB_N1_M5_Time_Scheduled;
	fbM6_OverallEquipmentEffectivenessOEE: FB_N1_M6_OverallEquipmentEffectivenessOEE;
	fbM7_MachineLearningCalculationDuration: FB_N1_M7_MachineLearningCalculationDuration;
	//SubNetworks
	fbN2_Products_Produced: FB_N2_Products_Produced;
	fbN3_Products_Defective: FB_N3_Products_Defective;
END_VAR

METHOD Call : BOOL
VAR_INPUT
	pAnalysis: POINTER TO FB_Analysis;
END_VAR
VAR
END_VAR

ValueMapping(pAnalysis);

//New Lambda Function
fbM1_State_Unit.Call(pAnalysis^.nContext);

//The Timing Analysis 1Ch measures time difference between on- and off-periods and counts the amount of on-periods. The on-period starts when the condition of operator and threshold is met. Optional a boolean signal for Enable Execution can be selected, so that the algorithm is just active if the value of the selected signal is TRUE.
fbM2_State_Execute.Call(pAnalysis^.nContext);

//The Timing Analysis 1Ch measures time difference between on- and off-periods and counts the amount of on-periods. The on-period starts when the condition of operator and threshold is met. Optional a boolean signal for Enable Execution can be selected, so that the algorithm is just active if the value of the selected signal is TRUE.
fbM3_State_Aborted.Call(pAnalysis^.nContext);

//The Timing Analysis 1Ch measures time difference between on- and off-periods and counts the amount of on-periods. The on-period starts when the condition of operator and threshold is met. Optional a boolean signal for Enable Execution can be selected, so that the algorithm is just active if the value of the selected signal is TRUE.
fbM4_State_Stopped.Call(pAnalysis^.nContext);

//The Timespan Operation executes a mathematical operation on two or more different input timespans and provides the result of the mathematical operation. The operator can be configured individually. Optional a boolean signal for Enable Execution can be selected, so that the algorithm is just active if the value of the selected signal is TRUE.
fbM5_Time_Scheduled.nTimeInCh1:= fbM2_State_Execute.fbTimeOnTotal.nRaw;
fbM5_Time_Scheduled.nTimeInCh2:= fbM3_State_Aborted.fbTimeOnTotal.nRaw;
fbM5_Time_Scheduled.nTimeInCh3:= fbM4_State_Stopped.fbTimeOnTotal.nRaw;
fbM5_Time_Scheduled.Call(pAnalysis^.nContext);

//Analytics Network "Products_Produced" with ID: 2
fbN2_Products_Produced.Call(pAnalysis);

//Analytics Network "Products_Defective" with ID: 3
fbN3_Products_Defective.Call(pAnalysis);

//The Overall Equipment Effectiveness (OEE) algorithm calculates key values to compare the current manufacturing process with its full potential. Optional a boolean signal for Enable Execution can be selected, so that the algorithm is just active if the value of the selected signal is TRUE.
fbM6_OverallEquipmentEffectivenessOEE.tScheduledTime:= fbM5_Time_Scheduled.fbTimespanResult.nRaw;
fbM6_OverallEquipmentEffectivenessOEE.tOperatingTime:= fbM2_State_Execute.fbTimeOnTotal.nRaw;
fbM6_OverallEquipmentEffectivenessOEE.nUnitsProduced:= fbN2_Products_Produced.nTotalCount;
fbM6_OverallEquipmentEffectivenessOEE.nDefectiveUnits:= fbN3_Products_Defective.nTotalCount;
fbM6_OverallEquipmentEffectivenessOEE.Call(pAnalysis^.nContext);

//The Min Max Avg 1Ch calculates minimum, maximum and average values of the input values from the beginning of the analysis up to the current moment. Furthermore the time values of the minimum and maximum are shown. Optional a boolean signal for Enable Execution can be selected, so that the algorithm is just active if the value of the selected signal is TRUE.
fbM7_MachineLearningCalculationDuration.Call(pAnalysis^.nContext);


//Error Handling
IF fbM1_State_Unit.bError THEN
	bError:= TRUE;
	ipTcResult:= fbM1_State_Unit.ipTcResult;
ELSIF fbM2_State_Execute.bError THEN
	bError:= TRUE;
	ipTcResult:= fbM2_State_Execute.ipTcResult;
ELSIF fbM3_State_Aborted.bError THEN
	bError:= TRUE;
	ipTcResult:= fbM3_State_Aborted.ipTcResult;
ELSIF fbM4_State_Stopped.bError THEN
	bError:= TRUE;
	ipTcResult:= fbM4_State_Stopped.ipTcResult;
ELSIF fbM5_Time_Scheduled.bError THEN
	bError:= TRUE;
	ipTcResult:= fbM5_Time_Scheduled.ipTcResult;
ELSIF fbN2_Products_Produced.bError THEN
	bError:= TRUE;
	ipTcResult:= fbN2_Products_Produced.ipTcResult;
ELSIF fbN3_Products_Defective.bError THEN
	bError:= TRUE;
	ipTcResult:= fbN3_Products_Defective.ipTcResult;
ELSIF fbM6_OverallEquipmentEffectivenessOEE.bError THEN
	bError:= TRUE;
	ipTcResult:= fbM6_OverallEquipmentEffectivenessOEE.ipTcResult;
ELSIF fbM7_MachineLearningCalculationDuration.bError THEN
	bError:= TRUE;
	ipTcResult:= fbM7_MachineLearningCalculationDuration.ipTcResult;
ELSE
	bError:= FALSE;
	ipTcResult:= fbTcMsgSuccess;
END_IF
END_METHOD

METHOD Reset : BOOL
VAR
	bResult: BOOL := TRUE;
END_VAR
bResult:= bResult AND fbM1_State_Unit.Reset();
bResult:= bResult AND fbM2_State_Execute.Reset();
bResult:= bResult AND fbM3_State_Aborted.Reset();
bResult:= bResult AND fbM4_State_Stopped.Reset();
bResult:= bResult AND fbM5_Time_Scheduled.Reset();
bResult:= bResult AND fbN2_Products_Produced.Reset();
bResult:= bResult AND fbN3_Products_Defective.Reset();
bResult:= bResult AND fbM6_OverallEquipmentEffectivenessOEE.Reset();
bResult:= bResult AND fbM7_MachineLearningCalculationDuration.Reset();
Reset:= bResult;
END_METHOD

METHOD PRIVATE ValueMapping : BOOL
VAR_INPUT
	pAnalysis: POINTER TO FB_Analysis;
END_VAR
VAR
END_VAR

//Module fbM1_State_Unit
fbM1_State_Unit.tTimestamp:= pAnalysis^.ipVirtual_Input_Source.tTimestamp;
fbM1_State_Unit.nInput:= pAnalysis^.ipVirtual_Input_Source.nV1_nState;


//Module fbM2_State_Execute
fbM2_State_Execute.tTimestamp:= pAnalysis^.ipVirtual_Input_Source.tTimestamp;
fbM2_State_Execute.nDataIn:= pAnalysis^.ipVirtual_Input_Source.nV1_nState;


//Module fbM3_State_Aborted
fbM3_State_Aborted.tTimestamp:= pAnalysis^.ipVirtual_Input_Source.tTimestamp;
fbM3_State_Aborted.nDataIn:= pAnalysis^.ipVirtual_Input_Source.nV1_nState;


//Module fbM4_State_Stopped
fbM4_State_Stopped.tTimestamp:= pAnalysis^.ipVirtual_Input_Source.tTimestamp;
fbM4_State_Stopped.nDataIn:= pAnalysis^.ipVirtual_Input_Source.nV1_nState;


//Module fbM6_OverallEquipmentEffectivenessOEE
fbM6_OverallEquipmentEffectivenessOEE.tTimestamp:= pAnalysis^.ipVirtual_Input_Source.tTimestamp;

//Module fbM7_MachineLearningCalculationDuration
fbM7_MachineLearningCalculationDuration.tTimestamp:= pAnalysis^.ipVirtual_Input_Source.tTimestamp;
fbM7_MachineLearningCalculationDuration.nDataIn:= pAnalysis^.ipVirtual_Input_Source.nV1_tMlCalculation;
END_METHOD

END_FUNCTION_BLOCK

// ---- POUs/Analytics/Analysis/Networks/N01 OEEDashboard/Modules/FB_N1_M1_State_Unit.TcPOU
//New Lambda Function
FUNCTION_BLOCK FB_N1_M1_State_Unit
VAR_INPUT
	nInput: UINT; 
	bEnableExecution: BOOL := TRUE; 
	tTimestamp: ULINT; 
	bReset: BOOL; 
	bReconfigure: BOOL := TRUE;
	sString0: STRING(255); 
	sString1: STRING(255); 
	sString2: STRING(255); 
	sString3: STRING(255); 
	sString4: STRING(255); 
	sString5: STRING(255); 
	sString6: STRING(255); 
	sString7: STRING(255); 
	sString8: STRING(255); 
	sString9: STRING(255); 
	sString10: STRING(255); 
	sString11: STRING(255); 
	sString12: STRING(255); 
	sString13: STRING(255); 
	sString14: STRING(255); 
	sString15: STRING(255); 
	sString16: STRING(255); 
	sString17: STRING(255); 
	sString18: STRING(255); 
	sString19: STRING(255); 
END_VAR
VAR_OUTPUT
	bError: BOOL;
	ipTcResult: I_TcMessage;
	sOutput: STRING(255);
	bNewResult: BOOL;
END_VAR
VAR
	bConfigured: BOOL;
	R_TRIG_Reconfigure: R_TRIG;
	
	fbL1_Lf_CppModuleAssignString: FB_L1_Lf_CppModuleAssignString(nObjID:=16#01010120);
END_VAR

METHOD Call : BOOL
VAR_INPUT
	nCurrentContext: DWORD;
END_VAR
VAR
END_VAR
IF NOT bConfigured THEN
	bConfigured:= TRUE;

	sString0:= 'Undefined';
	sString1:= 'Clearing';
	sString2:= 'Stopped';
	sString3:= 'Starting';
	sString4:= 'Idle';
	sString5:= 'Suspended';
	sString6:= 'Execute';
	sString7:= 'Stopping';
	sString8:= 'Aborting';
	sString9:= 'Aborted';
	sString10:= 'Holding';
	sString11:= 'Held';
	sString12:= 'Unholding';
	sString13:= 'Suspending';
	sString14:= 'Unsuspending';
	sString15:= 'Resetting';
	sString16:= 'Completing';
	sString17:= 'Complete';
	sString18:= '';
	sString19:= '';
END_IF

R_TRIG_Reconfigure(CLK:= bReconfigure);
IF R_TRIG_Reconfigure.Q THEN
	fbL1_Lf_CppModuleAssignString.SetInitValues(
		nInput:= nInput,
		ntTimestamp:= tTimestamp,
		bReset:= bReset,
		bEnableExecution:= bEnableExecution,
		pString0:= ADR(sString0),
		pString1:= ADR(sString1),
		pString2:= ADR(sString2),
		pString3:= ADR(sString3),
		pString4:= ADR(sString4),
		pString5:= ADR(sString5),
		pString6:= ADR(sString6),
		pString7:= ADR(sString7),
		pString8:= ADR(sString8),
		pString9:= ADR(sString9),
		pString10:= ADR(sString10),
		pString11:= ADR(sString11),
		pString12:= ADR(sString12),
		pString13:= ADR(sString13),
		pString14:= ADR(sString14),
		pString15:= ADR(sString15),
		pString16:= ADR(sString16),
		pString17:= ADR(sString17),
		pString18:= ADR(sString18),
		pString19:= ADR(sString19));

	bReconfigure:= FALSE;
END_IF

IF bReset THEN
	Reset();
END_IF

IF bEnableExecution THEN
	IF F_HasContext(nCurrentContext, nContext) THEN
		fbL1_Lf_CppModuleAssignString.SetValues(
			nInput:= nInput,
			ntTimestamp:= tTimestamp,
			bReset:= bReset,
			bEnableExecution:= bEnableExecution,
			pString0:= ADR(sString0),
			pString1:= ADR(sString1),
			pString2:= ADR(sString2),
			pString3:= ADR(sString3),
			pString4:= ADR(sString4),
			pString5:= ADR(sString5),
			pString6:= ADR(sString6),
			pString7:= ADR(sString7),
			pString8:= ADR(sString8),
			pString9:= ADR(sString9),
			pString10:= ADR(sString10),
			pString11:= ADR(sString11),
			pString12:= ADR(sString12),
			pString13:= ADR(sString13),
			pString14:= ADR(sString14),
			pString15:= ADR(sString15),
			pString16:= ADR(sString16),
			pString17:= ADR(sString17),
			pString18:= ADR(sString18),
			pString19:= ADR(sString19));

		fbL1_Lf_CppModuleAssignString.Call();

		fbL1_Lf_CppModuleAssignString.GetResults(
			pOutput:= ADR(sOutput),
			pbNewResult:= ADR(bNewResult),
			pString0:= ADR(sString0),
			pString1:= ADR(sString1),
			pString2:= ADR(sString2),
			pString3:= ADR(sString3),
			pString4:= ADR(sString4),
			pString5:= ADR(sString5),
			pString6:= ADR(sString6),
			pString7:= ADR(sString7),
			pString8:= ADR(sString8),
			pString9:= ADR(sString9),
			pString10:= ADR(sString10),
			pString11:= ADR(sString11),
			pString12:= ADR(sString12),
			pString13:= ADR(sString13),
			pString14:= ADR(sString14),
			pString15:= ADR(sString15),
			pString16:= ADR(sString16),
			pString17:= ADR(sString17),
			pString18:= ADR(sString18),
			pString19:= ADR(sString19));

		bNewResult:= fbL1_Lf_CppModuleAssignString.bNewResult;
		bError:= fbL1_Lf_CppModuleAssignString.bError;
		ipTcResult:= fbL1_Lf_CppModuleAssignString.ipTcResult;
	END_IF
ELSE
	bNewResult:= FALSE;
END_IF
END_METHOD

METHOD Reset : BOOL
VAR
END_VAR
Reset:= fbL1_Lf_CppModuleAssignString.Reset();
END_METHOD

METHOD SetHMI : BOOL
VAR_INPUT
	nContent: DINT;
	pContent: PVOID;
	bHMIReinit: BOOL;
END_VAR
VAR
	pHMI_C1_OEE_Dashboard: POINTER TO ST_HMI_C1_OEE_Dashboard;
END_VAR
SetHMI:= FALSE;

CASE nContent OF
	1:
		pHMI_C1_OEE_Dashboard:= pContent;

		IF bHMIReinit AND bConfigured THEN
			SetHMI:= TRUE;
		END_IF

		pHMI_C1_OEE_Dashboard^.stHMI_C1_Ctrl3_State_Unit.sM1_sOutput:= sOutput;
END_CASE
END_METHOD

METHOD GetHMI : BOOL
VAR_INPUT
	nContent: DINT;
	pContent: PVOID;
END_VAR
VAR
	pHMI_C1_OEE_Dashboard: POINTER TO ST_HMI_C1_OEE_Dashboard;
END_VAR

CASE nContent OF
	1:
		//OEE_Dashboard
		pHMI_C1_OEE_Dashboard:= pContent;

		IF pHMI_C1_OEE_Dashboard^.stHMI_C1_Ctrl3_State_Unit.bTrigReconfigure THEN
			pHMI_C1_OEE_Dashboard^.stHMI_C1_Ctrl3_State_Unit.bTrigReconfigure:= FALSE;
			bReconfigure:= TRUE;

		END_IF
END_CASE

GetHMI:= bReconfigure;
END_METHOD

PROPERTY nContext : DWORD
GET
nContext:= E_VirtualInput.eContext_V1_Virtual_Input_Source;
END_GET
END_PROPERTY

END_FUNCTION_BLOCK

// ---- POUs/Analytics/Lambda/FB_L1_Lf_CppModuleAssignString.TcPOU
FUNCTION_BLOCK FB_L1_Lf_CppModuleAssignString
VAR_OUTPUT
	bError: BOOL;
	ipTcResult: I_TcMessage := fbTcMessage;
	bNewResult: BOOL;
END_VAR
VAR
	hr: HRESULT;
	stEventEntry: TcEventEntry;
	
	fbTcMessage: FB_TcMessage;
	fbSrceInfo: FB_TcSourceInfo;
	
	ipLambda: ILf_CppModuleAssignString;
	iidLambda: IID := TC_GLOBAL_IID_LIST.IID_ILf_CppModuleAssignString;
END_VAR

//returns TRUE if succeeded
METHOD Call : BOOL
VAR
END_VAR
IF ipLambda <> 0 THEN
	hr:= ipLambda.Call();

	bError:= FAILED(hr);
	IF HRESULTAdsErr_TO_TcEventEntry(hr, stEventEntry) THEN
		fbTcMessage.CreateEx(stEventEntry, fbSrceInfo);
	END_IF

	bNewResult:= FALSE;

	Call:= NOT bError;
END_IF
END_METHOD

METHOD CreateInstance : BOOL
VAR_INPUT
	nObjID: OTCID;
END_VAR
VAR
END_VAR
IF ipLambda = 0 THEN
	IF nObjID <> 0 THEN
		hr:= FW_ObjMgr_GetObjectInstance(oid:=nObjID, iid:=iidLambda, pipUnk:=ADR(ipLambda));
	ELSE
		hr:= E_HRESULTAdsErr.INVALIDOBJID;
	END_IF

	bError:= FAILED(hr);
	IF HRESULTAdsErr_TO_TcEventEntry(hr, stEventEntry) THEN
		fbTcMessage.CreateEx(stEventEntry, fbSrceInfo);
	END_IF
END_IF
END_METHOD

METHOD FB_exit : BOOL
VAR_INPUT
	bInCopyCode: BOOL; // if TRUE, the exit method is called for exiting an instance that is copied afterwards (online change).
END_VAR
VAR
END_VAR
IF NOT bInCopyCode THEN //if not online change
	FW_SafeRelease(ADR(ipLambda));
END_IF
END_METHOD

METHOD FB_init : BOOL
VAR_INPUT
	bInitRetains: BOOL; // if TRUE, the retain variables are initialized (warm start / cold start)
	bInCopyCode: BOOL; // if TRUE, the instance afterwards gets moved into the copy code (online change)
	nObjID: OTCID;
END_VAR
VAR
END_VAR
IF NOT bInCopyCode THEN //if not online change
	IF nObjID <> 0 THEN
		CreateInstance(nObjID:= nObjID);
	END_IF
END_IF
END_METHOD

//returns TRUE if succeeded
METHOD GetResults : BOOL
VAR_INPUT
	pOutput: POINTER TO STRING(255);
	pbNewResult: POINTER TO BOOL;
	pString0: POINTER TO STRING(255);
	pString1: POINTER TO STRING(255);
	pString2: POINTER TO STRING(255);
	pString3: POINTER TO STRING(255);
	pString4: POINTER TO STRING(255);
	pString5: POINTER TO STRING(255);
	pString6: POINTER TO STRING(255);
	pString7: POINTER TO STRING(255);
	pString8: POINTER TO STRING(255);
	pString9: POINTER TO STRING(255);
	pString10: POINTER TO STRING(255);
	pString11: POINTER TO STRING(255);
	pString12: POINTER TO STRING(255);
	pString13: POINTER TO STRING(255);
	pString14: POINTER TO STRING(255);
	pString15: POINTER TO STRING(255);
	pString16: POINTER TO STRING(255);
	pString17: POINTER TO STRING(255);
	pString18: POINTER TO STRING(255);
	pString19: POINTER TO STRING(255);
END_VAR
VAR
END_VAR
IF ipLambda <> 0 THEN
	hr:= ipLambda.GetResults(
	Output:= pOutput,
	bNewResult:= pbNewResult,
	String0:= pString0,
	String1:= pString1,
	String2:= pString2,
	String3:= pString3,
	String4:= pString4,
	String5:= pString5,
	String6:= pString6,
	String7:= pString7,
	String8:= pString8,
	String9:= pString9,
	String10:= pString10,
	String11:= pString11,
	String12:= pString12,
	String13:= pString13,
	String14:= pString14,
	String15:= pString15,
	String16:= pString16,
	String17:= pString17,
	String18:= pString18,
	String19:= pString19);

	bError:= FAILED(hr);
	IF HRESULTAdsErr_TO_TcEventEntry(hr, stEventEntry) THEN
		fbTcMessage.CreateEx(stEventEntry, fbSrceInfo);
	END_IF

	bNewResult:= NOT bError;

	GetResults:= NOT bError;
END_IF
END_METHOD

//returns TRUE if succeeded
METHOD Reset : BOOL
VAR
END_VAR
IF ipLambda <> 0 THEN
	hr:= ipLambda.Reset();

	bError:= FAILED(hr);
	IF HRESULTAdsErr_TO_TcEventEntry(hr, stEventEntry) THEN
		fbTcMessage.CreateEx(stEventEntry, fbSrceInfo);
	END_IF

	Reset:= NOT bError;
END_IF
END_METHOD

//returns TRUE if succeeded
METHOD SetInitValues : BOOL
VAR_INPUT
	nInput: UINT;
	ntTimestamp: ULINT;
	bReset: BOOL;
	bEnableExecution: BOOL;
	pString0: POINTER TO STRING(255);
	pString1: POINTER TO STRING(255);
	pString2: POINTER TO STRING(255);
	pString3: POINTER TO STRING(255);
	pString4: POINTER TO STRING(255);
	pString5: POINTER TO STRING(255);
	pString6: POINTER TO STRING(255);
	pString7: POINTER TO STRING(255);
	pString8: POINTER TO STRING(255);
	pString9: POINTER TO STRING(255);
	pString10: POINTER TO STRING(255);
	pString11: POINTER TO STRING(255);
	pString12: POINTER TO STRING(255);
	pString13: POINTER TO STRING(255);
	pString14: POINTER TO STRING(255);
	pString15: POINTER TO STRING(255);
	pString16: POINTER TO STRING(255);
	pString17: POINTER TO STRING(255);
	pString18: POINTER TO STRING(255);
	pString19: POINTER TO STRING(255);
END_VAR
VAR
END_VAR
IF ipLambda <> 0 THEN
	hr:= ipLambda.SetInitValues(
	Input:= nInput,
	tTimestamp:= ntTimestamp,
	bReset:= bReset,
	bEnableExecution:= bEnableExecution,
	String0:= pString0,
	String1:= pString1,
	String2:= pString2,
	String3:= pString3,
	String4:= pString4,
	String5:= pString5,
	String6:= pString6,
	String7:= pString7,
	String8:= pString8,
	String9:= pString9,
	String10:= pString10,
	String11:= pString11,
	String12:= pString12,
	String13:= pString13,
	String14:= pString14,
	String15:= pString15,
	String16:= pString16,
	String17:= pString17,
	String18:= pString18,
	String19:= pString19);

	bError:= FAILED(hr);
	IF HRESULTAdsErr_TO_TcEventEntry(hr, stEventEntry) THEN
		fbTcMessage.CreateEx(stEventEntry, fbSrceInfo);
	END_IF

	SetInitValues:= NOT bError;
END_IF
END_METHOD

//returns TRUE if succeeded
METHOD SetValues : BOOL
VAR_INPUT
	nInput: UINT;
	ntTimestamp: ULINT;
	bReset: BOOL;
	bEnableExecution: BOOL;
	pString0: POINTER TO STRING(255);
	pString1: POINTER TO STRING(255);
	pString2: POINTER TO STRING(255);
	pString3: POINTER TO STRING(255);
	pString4: POINTER TO STRING(255);
	pString5: POINTER TO STRING(255);
	pString6: POINTER TO STRING(255);
	pString7: POINTER TO STRING(255);
	pString8: POINTER TO STRING(255);
	pString9: POINTER TO STRING(255);
	pString10: POINTER TO STRING(255);
	pString11: POINTER TO STRING(255);
	pString12: POINTER TO STRING(255);
	pString13: POINTER TO STRING(255);
	pString14: POINTER TO STRING(255);
	pString15: POINTER TO STRING(255);
	pString16: POINTER TO STRING(255);
	pString17: POINTER TO STRING(255);
	pString18: POINTER TO STRING(255);
	pString19: POINTER TO STRING(255);
END_VAR
VAR
END_VAR
IF ipLambda <> 0 THEN
	hr:= ipLambda.SetValues(
	Input:= nInput,
	tTimestamp:= ntTimestamp,
	bReset:= bReset,
	bEnableExecution:= bEnableExecution,
	String0:= pString0,
	String1:= pString1,
	String2:= pString2,
	String3:= pString3,
	String4:= pString4,
	String5:= pString5,
	String6:= pString6,
	String7:= pString7,
	String8:= pString8,
	String9:= pString9,
	String10:= pString10,
	String11:= pString11,
	String12:= pString12,
	String13:= pString13,
	String14:= pString14,
	String15:= pString15,
	String16:= pString16,
	String17:= pString17,
	String18:= pString18,
	String19:= pString19);

	bError:= FAILED(hr);
	IF HRESULTAdsErr_TO_TcEventEntry(hr, stEventEntry) THEN
		fbTcMessage.CreateEx(stEventEntry, fbSrceInfo);
	END_IF

	SetValues:= NOT bError;
END_IF
END_METHOD

END_FUNCTION_BLOCK

// ---- POUs/Analytics/[Helper]/F_HasContext.TcPOU
FUNCTION F_HasContext : BOOL
VAR_INPUT
	nContext: DWORD;
	nSearchContext: DWORD;
END_VAR
VAR
END_VAR


F_HasContext:= (nContext > 0) AND (((nContext AND nSearchContext) > 0) OR (nSearchContext = E_DataSourceContext.eContext_Unknown));

END_FUNCTION

// ---- POUs/Analytics/Analysis/Networks/N01 OEEDashboard/Modules/FB_N1_M2_State_Execute.TcPOU
//The Timing Analysis 1Ch measures time difference between on- and off-periods and counts the amount of on-periods. The on-period starts when the condition of operator and threshold is met. Optional a boolean signal for Enable Execution can be selected, so that the algorithm is just active if the value of the selected signal is TRUE.
FUNCTION_BLOCK FB_N1_M2_State_Execute
VAR_INPUT
	nDataIn: UINT; 
	tTimestamp: ULINT; 
	bEnableExecution: BOOL := TRUE; 
	bReset: BOOL; 
	bReconfigure: BOOL := TRUE;
END_VAR
VAR_INPUT PERSISTENT
	stThresholdLevelOn: ST_ALY_Threshold; 
	fTolerance: LREAL; 
END_VAR
VAR_OUTPUT
	bError: BOOL;
	ipTcResult: I_TcMessage;
	bNewResult: BOOL;
	bIsOn: BOOL;
	nCountOn: ULINT;
	fbTimeCurrentInterval: FB_ALY_TimeSpan;
	fbTimeOnTotal: FB_ALY_TimeSpan;
	fbTimeOffTotal: FB_ALY_TimeSpan;
END_VAR
VAR
	
	R_TRIG_Reconfigure: R_TRIG;
	
	fbALY_TimingAnalysis_1Ch: FB_ALY_TimingAnalysis_1Ch := ( bPersistent:= TRUE );
END_VAR
VAR PERSISTENT
	bConfigured: BOOL;
END_VAR

METHOD Call : BOOL
VAR_INPUT
	nCurrentContext: DWORD;
END_VAR
VAR
END_VAR
IF NOT bConfigured THEN
	bConfigured:= TRUE;

	fTolerance:= 0;

	stThresholdLevelOn.eComparisonOperator:= E_ALY_ComparisonOperator.Equals;
	stThresholdLevelOn.fThreshold:= 6;

	fbALY_TimingAnalysis_1Ch.fTolerance:= fTolerance;
END_IF

R_TRIG_Reconfigure(CLK:= bReconfigure);
IF R_TRIG_Reconfigure.Q THEN
	fbALY_TimingAnalysis_1Ch.ConfigureChannel(stThresholdLevel:= stThresholdLevelOn);

	fbALY_TimingAnalysis_1Ch.Configure();

	bReconfigure:= FALSE;
END_IF

IF bReset THEN
	Reset();
END_IF

IF bEnableExecution THEN
	IF F_HasContext(nCurrentContext, nContext) THEN
		fbALY_TimingAnalysis_1Ch.SetChannelValue(Input:= nDataIn);

		fbALY_TimingAnalysis_1Ch.Call(tTimestamp:= tTimestamp);

		bNewResult:= fbALY_TimingAnalysis_1Ch.bNewResult;
		bIsOn:= fbALY_TimingAnalysis_1Ch.bIsOn;
		nCountOn:= fbALY_TimingAnalysis_1Ch.nCountOn;
		fbTimeCurrentInterval:= fbALY_TimingAnalysis_1Ch.fbTimeCurrentInterval;
		fbTimeOnTotal:= fbALY_TimingAnalysis_1Ch.fbTimeOnTotal;
		fbTimeOffTotal:= fbALY_TimingAnalysis_1Ch.fbTimeOffTotal;

		bError:= fbALY_TimingAnalysis_1Ch.bError;
		ipTcResult:= fbALY_TimingAnalysis_1Ch.ipResultMessage;
	END_IF
ELSE
	bNewResult:= FALSE;
END_IF
END_METHOD

METHOD Reset : BOOL
VAR
END_VAR
Reset:= fbALY_TimingAnalysis_1Ch.Reset();

bNewResult:= fbALY_TimingAnalysis_1Ch.bNewResult;
bIsOn:= fbALY_TimingAnalysis_1Ch.bIsOn;
nCountOn:= fbALY_TimingAnalysis_1Ch.nCountOn;
fbTimeCurrentInterval:= fbALY_TimingAnalysis_1Ch.fbTimeCurrentInterval;
fbTimeOnTotal:= fbALY_TimingAnalysis_1Ch.fbTimeOnTotal;
fbTimeOffTotal:= fbALY_TimingAnalysis_1Ch.fbTimeOffTotal;

bError:= NOT Reset;
ipTcResult:= fbALY_TimingAnalysis_1Ch.ipResultMessage;
END_METHOD

PROPERTY nContext : DWORD
GET
nContext:= E_VirtualInput.eContext_V1_Virtual_Input_Source;
END_GET
END_PROPERTY

END_FUNCTION_BLOCK

// ---- POUs/Analytics/Analysis/Networks/N01 OEEDashboard/Modules/FB_N1_M3_State_Aborted.TcPOU
//The Timing Analysis 1Ch measures time difference between on- and off-periods and counts the amount of on-periods. The on-period starts when the condition of operator and threshold is met. Optional a boolean signal for Enable Execution can be selected, so that the algorithm is just active if the value of the selected signal is TRUE.
FUNCTION_BLOCK FB_N1_M3_State_Aborted
VAR_INPUT
	nDataIn: UINT; 
	tTimestamp: ULINT; 
	bEnableExecution: BOOL := TRUE; 
	bReset: BOOL; 
	bReconfigure: BOOL := TRUE;
END_VAR
VAR_INPUT PERSISTENT
	stThresholdLevelOn: ST_ALY_Threshold; 
	fTolerance: LREAL; 
END_VAR
VAR_OUTPUT
	bError: BOOL;
	ipTcResult: I_TcMessage;
	bNewResult: BOOL;
	bIsOn: BOOL;
	nCountOn: ULINT;
	fbTimeCurrentInterval: FB_ALY_TimeSpan;
	fbTimeOnTotal: FB_ALY_TimeSpan;
	fbTimeOffTotal: FB_ALY_TimeSpan;
END_VAR
VAR
	
	R_TRIG_Reconfigure: R_TRIG;
	
	fbALY_TimingAnalysis_1Ch: FB_ALY_TimingAnalysis_1Ch := ( bPersistent:= TRUE );
END_VAR
VAR PERSISTENT
	bConfigured: BOOL;
END_VAR

METHOD Call : BOOL
VAR_INPUT
	nCurrentContext: DWORD;
END_VAR
VAR
END_VAR
IF NOT bConfigured THEN
	bConfigured:= TRUE;

	fTolerance:= 0;

	stThresholdLevelOn.eComparisonOperator:= E_ALY_ComparisonOperator.Equals;
	stThresholdLevelOn.fThreshold:= 9;

	fbALY_TimingAnalysis_1Ch.fTolerance:= fTolerance;
END_IF

R_TRIG_Reconfigure(CLK:= bReconfigure);
IF R_TRIG_Reconfigure.Q THEN
	fbALY_TimingAnalysis_1Ch.ConfigureChannel(stThresholdLevel:= stThresholdLevelOn);

	fbALY_TimingAnalysis_1Ch.Configure();

	bReconfigure:= FALSE;
END_IF

IF bReset THEN
	Reset();
END_IF

IF bEnableExecution THEN
	IF F_HasContext(nCurrentContext, nContext) THEN
		fbALY_TimingAnalysis_1Ch.SetChannelValue(Input:= nDataIn);

		fbALY_TimingAnalysis_1Ch.Call(tTimestamp:= tTimestamp);

		bNewResult:= fbALY_TimingAnalysis_1Ch.bNewResult;
		bIsOn:= fbALY_TimingAnalysis_1Ch.bIsOn;
		nCountOn:= fbALY_TimingAnalysis_1Ch.nCountOn;
		fbTimeCurrentInterval:= fbALY_TimingAnalysis_1Ch.fbTimeCurrentInterval;
		fbTimeOnTotal:= fbALY_TimingAnalysis_1Ch.fbTimeOnTotal;
		fbTimeOffTotal:= fbALY_TimingAnalysis_1Ch.fbTimeOffTotal;

		bError:= fbALY_TimingAnalysis_1Ch.bError;
		ipTcResult:= fbALY_TimingAnalysis_1Ch.ipResultMessage;
	END_IF
ELSE
	bNewResult:= FALSE;
END_IF
END_METHOD

METHOD Reset : BOOL
VAR
END_VAR
Reset:= fbALY_TimingAnalysis_1Ch.Reset();

bNewResult:= fbALY_TimingAnalysis_1Ch.bNewResult;
bIsOn:= fbALY_TimingAnalysis_1Ch.bIsOn;
nCountOn:= fbALY_TimingAnalysis_1Ch.nCountOn;
fbTimeCurrentInterval:= fbALY_TimingAnalysis_1Ch.fbTimeCurrentInterval;
fbTimeOnTotal:= fbALY_TimingAnalysis_1Ch.fbTimeOnTotal;
fbTimeOffTotal:= fbALY_TimingAnalysis_1Ch.fbTimeOffTotal;

bError:= NOT Reset;
ipTcResult:= fbALY_TimingAnalysis_1Ch.ipResultMessage;
END_METHOD

PROPERTY nContext : DWORD
GET
nContext:= E_VirtualInput.eContext_V1_Virtual_Input_Source;
END_GET
END_PROPERTY

END_FUNCTION_BLOCK

// ---- POUs/Analytics/Analysis/Networks/N01 OEEDashboard/Modules/FB_N1_M4_State_Stopped.TcPOU
//The Timing Analysis 1Ch measures time difference between on- and off-periods and counts the amount of on-periods. The on-period starts when the condition of operator and threshold is met. Optional a boolean signal for Enable Execution can be selected, so that the algorithm is just active if the value of the selected signal is TRUE.
FUNCTION_BLOCK FB_N1_M4_State_Stopped
VAR_INPUT
	nDataIn: UINT; 
	tTimestamp: ULINT; 
	bEnableExecution: BOOL := TRUE; 
	bReset: BOOL; 
	bReconfigure: BOOL := TRUE;
END_VAR
VAR_INPUT PERSISTENT
	stThresholdLevelOn: ST_ALY_Threshold; 
	fTolerance: LREAL; 
END_VAR
VAR_OUTPUT
	bError: BOOL;
	ipTcResult: I_TcMessage;
	bNewResult: BOOL;
	bIsOn: BOOL;
	nCountOn: ULINT;
	fbTimeCurrentInterval: FB_ALY_TimeSpan;
	fbTimeOnTotal: FB_ALY_TimeSpan;
	fbTimeOffTotal: FB_ALY_TimeSpan;
END_VAR
VAR
	
	R_TRIG_Reconfigure: R_TRIG;
	
	fbALY_TimingAnalysis_1Ch: FB_ALY_TimingAnalysis_1Ch := ( bPersistent:= TRUE );
END_VAR
VAR PERSISTENT
	bConfigured: BOOL;
END_VAR

METHOD Call : BOOL
VAR_INPUT
	nCurrentContext: DWORD;
END_VAR
VAR
END_VAR
IF NOT bConfigured THEN
	bConfigured:= TRUE;

	fTolerance:= 0;

	stThresholdLevelOn.eComparisonOperator:= E_ALY_ComparisonOperator.Equals;
	stThresholdLevelOn.fThreshold:= 2;

	fbALY_TimingAnalysis_1Ch.fTolerance:= fTolerance;
END_IF

R_TRIG_Reconfigure(CLK:= bReconfigure);
IF R_TRIG_Reconfigure.Q THEN
	fbALY_TimingAnalysis_1Ch.ConfigureChannel(stThresholdLevel:= stThresholdLevelOn);

	fbALY_TimingAnalysis_1Ch.Configure();

	bReconfigure:= FALSE;
END_IF

IF bReset THEN
	Reset();
END_IF

IF bEnableExecution THEN
	IF F_HasContext(nCurrentContext, nContext) THEN
		fbALY_TimingAnalysis_1Ch.SetChannelValue(Input:= nDataIn);

		fbALY_TimingAnalysis_1Ch.Call(tTimestamp:= tTimestamp);

		bNewResult:= fbALY_TimingAnalysis_1Ch.bNewResult;
		bIsOn:= fbALY_TimingAnalysis_1Ch.bIsOn;
		nCountOn:= fbALY_TimingAnalysis_1Ch.nCountOn;
		fbTimeCurrentInterval:= fbALY_TimingAnalysis_1Ch.fbTimeCurrentInterval;
		fbTimeOnTotal:= fbALY_TimingAnalysis_1Ch.fbTimeOnTotal;
		fbTimeOffTotal:= fbALY_TimingAnalysis_1Ch.fbTimeOffTotal;

		bError:= fbALY_TimingAnalysis_1Ch.bError;
		ipTcResult:= fbALY_TimingAnalysis_1Ch.ipResultMessage;
	END_IF
ELSE
	bNewResult:= FALSE;
END_IF
END_METHOD

METHOD Reset : BOOL
VAR
END_VAR
Reset:= fbALY_TimingAnalysis_1Ch.Reset();

bNewResult:= fbALY_TimingAnalysis_1Ch.bNewResult;
bIsOn:= fbALY_TimingAnalysis_1Ch.bIsOn;
nCountOn:= fbALY_TimingAnalysis_1Ch.nCountOn;
fbTimeCurrentInterval:= fbALY_TimingAnalysis_1Ch.fbTimeCurrentInterval;
fbTimeOnTotal:= fbALY_TimingAnalysis_1Ch.fbTimeOnTotal;
fbTimeOffTotal:= fbALY_TimingAnalysis_1Ch.fbTimeOffTotal;

bError:= NOT Reset;
ipTcResult:= fbALY_TimingAnalysis_1Ch.ipResultMessage;
END_METHOD

PROPERTY nContext : DWORD
GET
nContext:= E_VirtualInput.eContext_V1_Virtual_Input_Source;
END_GET
END_PROPERTY

END_FUNCTION_BLOCK

// ---- POUs/Analytics/Analysis/Networks/N01 OEEDashboard/Modules/FB_N1_M5_Time_Scheduled.TcPOU
//The Timespan Operation executes a mathematical operation on two or more different input timespans and provides the result of the mathematical operation. The operator can be configured individually. Optional a boolean signal for Enable Execution can be selected, so that the algorithm is just active if the value of the selected signal is TRUE.
FUNCTION_BLOCK FB_N1_M5_Time_Scheduled
VAR_INPUT
	nTimeInCh1: LINT; 
	nTimeInCh2: LINT; 
	nTimeInCh3: LINT; 
	bEnableExecution: BOOL := TRUE; 
	bReset: BOOL; 
	bReconfigure: BOOL := TRUE;
END_VAR
VAR_INPUT PERSISTENT
	eTimespanOperator: E_ALY_TimespanOperator; 
END_VAR
VAR_OUTPUT
	bError: BOOL;
	ipTcResult: I_TcMessage;
	bNewResult: BOOL;
	fbTimespanResult: FB_ALY_TimeSpan;
END_VAR
VAR
	
	R_TRIG_Reconfigure: R_TRIG;
	
	fbALY_TimespanOperation: FB_ALY_TimespanOperation(nNumChannels:=3);
END_VAR
VAR PERSISTENT
	bConfigured: BOOL;
END_VAR

METHOD Call : BOOL
VAR_INPUT
	nCurrentContext: DWORD;
END_VAR
VAR
END_VAR
IF NOT bConfigured THEN
	bConfigured:= TRUE;

	eTimespanOperator:= E_ALY_TimespanOperator.Addition;

END_IF

R_TRIG_Reconfigure(CLK:= bReconfigure);
IF R_TRIG_Reconfigure.Q THEN
	fbALY_TimespanOperation.Configure(eTimespanOperator:= eTimespanOperator);

	bReconfigure:= FALSE;
END_IF

IF bReset THEN
	Reset();
END_IF

IF bEnableExecution THEN
	IF F_HasContext(nCurrentContext, nContext) THEN
		fbALY_TimespanOperation.SetChannelValue(nChannel:= 1, Input:= nTimeInCh1);
		fbALY_TimespanOperation.SetChannelValue(nChannel:= 2, Input:= nTimeInCh2);
		fbALY_TimespanOperation.SetChannelValue(nChannel:= 3, Input:= nTimeInCh3);

		fbALY_TimespanOperation.Call();


		bNewResult:= fbALY_TimespanOperation.bNewResult;
		fbTimespanResult:= fbALY_TimespanOperation.fbTimespanResult;

		bError:= fbALY_TimespanOperation.bError;
		ipTcResult:= fbALY_TimespanOperation.ipResultMessage;
	END_IF
ELSE
	bNewResult:= FALSE;
END_IF
END_METHOD

METHOD Reset : BOOL
VAR
END_VAR
Reset:= fbALY_TimespanOperation.Reset();

bNewResult:= fbALY_TimespanOperation.bNewResult;
fbTimespanResult:= fbALY_TimespanOperation.fbTimespanResult;

bError:= NOT Reset;
ipTcResult:= fbALY_TimespanOperation.ipResultMessage;
END_METHOD

PROPERTY nContext : DWORD
GET
nContext:= E_VirtualInput.eContext_V1_Virtual_Input_Source;
END_GET
END_PROPERTY

END_FUNCTION_BLOCK

// ---- POUs/Analytics/Analysis/Networks/N01 OEEDashboard/Modules/FB_N1_M6_OverallEquipmentEffectivenessOEE.TcPOU
//The Overall Equipment Effectiveness (OEE) algorithm calculates key values to compare the current manufacturing process with its full potential. Optional a boolean signal for Enable Execution can be selected, so that the algorithm is just active if the value of the selected signal is TRUE.
FUNCTION_BLOCK FB_N1_M6_OverallEquipmentEffectivenessOEE
VAR_INPUT
	tScheduledTime: LINT; 
	tOperatingTime: LINT; 
	nUnitsProduced: ULINT; 
	nDefectiveUnits: ULINT; 
	tTimestamp: ULINT; 
	bEnableExecution: BOOL := TRUE; 
	bReset: BOOL; 
	bReconfigure: BOOL := TRUE;
END_VAR
VAR_INPUT PERSISTENT
	tIdealCycleTime: LTIME; 
	fThresholdLevelOkWarning: LREAL; 
	fThresholdLevelWarningAlarm: LREAL; 
END_VAR
VAR_OUTPUT
	bError: BOOL;
	ipTcResult: I_TcMessage;
	bNewResult: BOOL;
	fOEE: LREAL;
	eOeeClass: E_ALY_Classification_3Cls;
	fAvailability: LREAL;
	fPerformance: LREAL;
	fQuality: LREAL;
	fbTimeOeeEventWarning: FB_ALY_DateTime;
	fbTimeOeeEventAlarm: FB_ALY_DateTime;
END_VAR
VAR
	
	R_TRIG_Reconfigure: R_TRIG;
	
	fbALY_OverallEquipmentEffectiveness: FB_ALY_OverallEquipmentEffectiveness;
END_VAR
VAR PERSISTENT
	bConfigured: BOOL;
END_VAR

METHOD Call : BOOL
VAR_INPUT
	nCurrentContext: DWORD;
END_VAR
VAR
END_VAR
IF NOT bConfigured THEN
	bConfigured:= TRUE;

	tIdealCycleTime:= LTIME#750000000ns;
	fThresholdLevelOkWarning:= 90;
	fThresholdLevelWarningAlarm:= 75;

END_IF

R_TRIG_Reconfigure(CLK:= bReconfigure);
IF R_TRIG_Reconfigure.Q THEN
	fbALY_OverallEquipmentEffectiveness.Configure(tIdealCycleTime:= tIdealCycleTime, fThresholdLevelOkWarning:= fThresholdLevelOkWarning, fThresholdLevelWarningAlarm:= fThresholdLevelWarningAlarm);

	bReconfigure:= FALSE;
END_IF

IF bReset THEN
	Reset();
END_IF

IF bEnableExecution THEN
	IF F_HasContext(nCurrentContext, nContext) THEN
		fbALY_OverallEquipmentEffectiveness.SetChannelValue(nChannel:= 1, Input:= tScheduledTime);
		fbALY_OverallEquipmentEffectiveness.SetChannelValue(nChannel:= 2, Input:= tOperatingTime);
		fbALY_OverallEquipmentEffectiveness.SetChannelValue(nChannel:= 3, Input:= nUnitsProduced);
		fbALY_OverallEquipmentEffectiveness.SetChannelValue(nChannel:= 4, Input:= nDefectiveUnits);

		fbALY_OverallEquipmentEffectiveness.Call(tTimestamp:= tTimestamp);

		bNewResult:= fbALY_OverallEquipmentEffectiveness.bNewResult;
		fOEE:= fbALY_OverallEquipmentEffectiveness.fOEE;
		eOeeClass:= fbALY_OverallEquipmentEffectiveness.eOeeClass;
		fAvailability:= fbALY_OverallEquipmentEffectiveness.fAvailability;
		fPerformance:= fbALY_OverallEquipmentEffectiveness.fPerformance;
		fQuality:= fbALY_OverallEquipmentEffectiveness.fQuality;
		fbTimeOeeEventWarning:= fbALY_OverallEquipmentEffectiveness.fbTimeOeeEventWarning;
		fbTimeOeeEventAlarm:= fbALY_OverallEquipmentEffectiveness.fbTimeOeeEventAlarm;

		bError:= fbALY_OverallEquipmentEffectiveness.bError;
		ipTcResult:= fbALY_OverallEquipmentEffectiveness.ipResultMessage;
	END_IF
ELSE
	bNewResult:= FALSE;
END_IF
END_METHOD

METHOD Reset : BOOL
VAR
END_VAR
Reset:= fbALY_OverallEquipmentEffectiveness.Reset();

bNewResult:= fbALY_OverallEquipmentEffectiveness.bNewResult;
fOEE:= fbALY_OverallEquipmentEffectiveness.fOEE;
eOeeClass:= fbALY_OverallEquipmentEffectiveness.eOeeClass;
fAvailability:= fbALY_OverallEquipmentEffectiveness.fAvailability;
fPerformance:= fbALY_OverallEquipmentEffectiveness.fPerformance;
fQuality:= fbALY_OverallEquipmentEffectiveness.fQuality;
fbTimeOeeEventWarning:= fbALY_OverallEquipmentEffectiveness.fbTimeOeeEventWarning;
fbTimeOeeEventAlarm:= fbALY_OverallEquipmentEffectiveness.fbTimeOeeEventAlarm;

bError:= NOT Reset;
ipTcResult:= fbALY_OverallEquipmentEffectiveness.ipResultMessage;
END_METHOD

METHOD SetHMI : BOOL
VAR_INPUT
	nContent: DINT;
	pContent: PVOID;
	bHMIReinit: BOOL;
END_VAR
VAR
	pHMI_C1_OEE_Dashboard: POINTER TO ST_HMI_C1_OEE_Dashboard;
END_VAR
SetHMI:= FALSE;

CASE nContent OF
	1:
		pHMI_C1_OEE_Dashboard:= pContent;

		IF bHMIReinit AND bConfigured THEN
			pHMI_C1_OEE_Dashboard^.stHMI_C1_Ctrl1_Overall_Equipment_Effectiveness_OEE.fM6_fThresholdLevelOkWarning:= fThresholdLevelOkWarning;
			pHMI_C1_OEE_Dashboard^.stHMI_C1_Ctrl1_Overall_Equipment_Effectiveness_OEE.fM6_fThresholdLevelWarningAlarm:= fThresholdLevelWarningAlarm;
			SetHMI:= TRUE;
		END_IF

		pHMI_C1_OEE_Dashboard^.stHMI_C1_Ctrl1_Overall_Equipment_Effectiveness_OEE.fM6_fOEE:= fOEE;
		pHMI_C1_OEE_Dashboard^.stHMI_C1_Ctrl1_Overall_Equipment_Effectiveness_OEE.fM6_fAvailability:= fAvailability;
		pHMI_C1_OEE_Dashboard^.stHMI_C1_Ctrl1_Overall_Equipment_Effectiveness_OEE.fM6_fPerformance:= fPerformance;
		pHMI_C1_OEE_Dashboard^.stHMI_C1_Ctrl1_Overall_Equipment_Effectiveness_OEE.fM6_fQuality:= fQuality;
		pHMI_C1_OEE_Dashboard^.stHMI_C1_Ctrl1_Overall_Equipment_Effectiveness_OEE.eM6_eOeeClass:= eOeeClass;
END_CASE
END_METHOD

METHOD GetHMI : BOOL
VAR_INPUT
	nContent: DINT;
	pContent: PVOID;
END_VAR
VAR
	pHMI_C1_OEE_Dashboard: POINTER TO ST_HMI_C1_OEE_Dashboard;
END_VAR

CASE nContent OF
	1:
		//OEE_Dashboard
		pHMI_C1_OEE_Dashboard:= pContent;

		IF pHMI_C1_OEE_Dashboard^.stHMI_C1_Ctrl1_Overall_Equipment_Effectiveness_OEE.bTrigReconfigure THEN
			pHMI_C1_OEE_Dashboard^.stHMI_C1_Ctrl1_Overall_Equipment_Effectiveness_OEE.bTrigReconfigure:= FALSE;
			bReconfigure:= TRUE;

			fThresholdLevelOkWarning:= pHMI_C1_OEE_Dashboard^.stHMI_C1_Ctrl1_Overall_Equipment_Effectiveness_OEE.fM6_fThresholdLevelOkWarning;
			fThresholdLevelWarningAlarm:= pHMI_C1_OEE_Dashboard^.stHMI_C1_Ctrl1_Overall_Equipment_Effectiveness_OEE.fM6_fThresholdLevelWarningAlarm;
		END_IF
END_CASE

GetHMI:= bReconfigure;
END_METHOD

PROPERTY nContext : DWORD
GET
nContext:= E_VirtualInput.eContext_V1_Virtual_Input_Source;
END_GET
END_PROPERTY

END_FUNCTION_BLOCK

// ---- POUs/Analytics/Analysis/Networks/N01 OEEDashboard/Modules/FB_N1_M7_MachineLearningCalculationDuration.TcPOU
//The Min Max Avg 1Ch calculates minimum, maximum and average values of the input values from the beginning of the analysis up to the current moment. Furthermore the time values of the minimum and maximum are shown. Optional a boolean signal for Enable Execution can be selected, so that the algorithm is just active if the value of the selected signal is TRUE.
FUNCTION_BLOCK FB_N1_M7_MachineLearningCalculationDuration
VAR_INPUT
	nDataIn: UDINT; 
	tTimestamp: ULINT; 
	bEnableExecution: BOOL := TRUE; 
	bReset: BOOL; 
END_VAR
VAR_OUTPUT
	bError: BOOL;
	ipTcResult: I_TcMessage;
	bNewResult: BOOL;
	fMin: LREAL;
	fMax: LREAL;
	fAvg: LREAL;
	fbTimeMin: FB_ALY_DateTime;
	fbTimeMax: FB_ALY_DateTime;
END_VAR
VAR
	
	
	fbALY_MinMaxAvg_1Ch: FB_ALY_MinMaxAvg_1Ch;
END_VAR

METHOD Call : BOOL
VAR_INPUT
	nCurrentContext: DWORD;
END_VAR
VAR
END_VAR
IF bReset THEN
	Reset();
END_IF

IF bEnableExecution THEN
	IF F_HasContext(nCurrentContext, nContext) THEN
		fbALY_MinMaxAvg_1Ch.SetChannelValue(Input:= nDataIn);

		fbALY_MinMaxAvg_1Ch.Call(tTimestamp:= tTimestamp);

		bNewResult:= fbALY_MinMaxAvg_1Ch.bNewResult;
		fMin:= fbALY_MinMaxAvg_1Ch.fMin;
		fMax:= fbALY_MinMaxAvg_1Ch.fMax;
		fAvg:= fbALY_MinMaxAvg_1Ch.fAvg;
		fbTimeMin:= fbALY_MinMaxAvg_1Ch.fbTimeMin;
		fbTimeMax:= fbALY_MinMaxAvg_1Ch.fbTimeMax;

		bError:= fbALY_MinMaxAvg_1Ch.bError;
		ipTcResult:= fbALY_MinMaxAvg_1Ch.ipResultMessage;
	END_IF
ELSE
	bNewResult:= FALSE;
END_IF
END_METHOD

METHOD Reset : BOOL
VAR
END_VAR
Reset:= fbALY_MinMaxAvg_1Ch.Reset();

bNewResult:= fbALY_MinMaxAvg_1Ch.bNewResult;
fMin:= fbALY_MinMaxAvg_1Ch.fMin;
fMax:= fbALY_MinMaxAvg_1Ch.fMax;
fAvg:= fbALY_MinMaxAvg_1Ch.fAvg;
fbTimeMin:= fbALY_MinMaxAvg_1Ch.fbTimeMin;
fbTimeMax:= fbALY_MinMaxAvg_1Ch.fbTimeMax;

bError:= NOT Reset;
ipTcResult:= fbALY_MinMaxAvg_1Ch.ipResultMessage;
END_METHOD

METHOD SetHMI : BOOL
VAR_INPUT
	nContent: DINT;
	pContent: PVOID;
	bHMIReinit: BOOL;
END_VAR
VAR
	pHMI_C1_OEE_Dashboard: POINTER TO ST_HMI_C1_OEE_Dashboard;
END_VAR
SetHMI:= FALSE;

CASE nContent OF
	1:
		pHMI_C1_OEE_Dashboard:= pContent;


		pHMI_C1_OEE_Dashboard^.stHMI_C1_Ctrl2_Machine_Learning_Calculation_Duration.nM7_nDataIn:= nDataIn;
		pHMI_C1_OEE_Dashboard^.stHMI_C1_Ctrl2_Machine_Learning_Calculation_Duration.fM7_fMin:= fMin;
		pHMI_C1_OEE_Dashboard^.stHMI_C1_Ctrl2_Machine_Learning_Calculation_Duration.fM7_fMax:= fMax;
		pHMI_C1_OEE_Dashboard^.stHMI_C1_Ctrl2_Machine_Learning_Calculation_Duration.fM7_fAvg:= fAvg;
		fbTimeMin.nUtcTimeBias:= -120; //UTC Offset [(UTC+01:00) Amsterdam, Berlin, Bern, Rome, Stockholm, Vienna]
		pHMI_C1_OEE_Dashboard^.stHMI_C1_Ctrl2_Machine_Learning_Calculation_Duration.tM7_fbTimeMin:= fbTimeMin.stStructured;
		fbTimeMax.nUtcTimeBias:= -120; //UTC Offset [(UTC+01:00) Amsterdam, Berlin, Bern, Rome, Stockholm, Vienna]
		pHMI_C1_OEE_Dashboard^.stHMI_C1_Ctrl2_Machine_Learning_Calculation_Duration.tM7_fbTimeMax:= fbTimeMax.stStructured;
END_CASE

SetHMI:= TRUE;
END_METHOD

METHOD GetHMI : BOOL
VAR_INPUT
	nContent: DINT;
	pContent: PVOID;
END_VAR
VAR
END_VAR
END_METHOD

PROPERTY nContext : DWORD
GET
nContext:= E_VirtualInput.eContext_V1_Virtual_Input_Source;
END_GET
END_PROPERTY

END_FUNCTION_BLOCK

// ---- POUs/Analytics/Analysis/Networks/N01 OEEDashboard/N02 Products_Produced/FB_N2_Products_Produced.TcPOU
//Analytics Network "Products_Produced" with ID: 2
{attribute 'no_assign'}
FUNCTION_BLOCK FB_N2_Products_Produced
VAR_INPUT
	nOngoingCount: ULINT;
END_VAR
VAR_OUTPUT
	bError: BOOL;
	ipTcResult: I_TcMessage := fbTcMsgSuccess;
	nTotalCount: ULINT;
END_VAR
VAR
	fbTcMsgSuccess: FB_TcMessageSuccess;
	
	//Modules
	fbM1_BatchNShift1Ch: FB_N2_M1_BatchNShift1Ch;
	fbM2_MathOperation: FB_N2_M2_MathOperation;
	fbM3_EdgeCounter1Ch: FB_N2_M3_EdgeCounter1Ch;
END_VAR

METHOD Call : BOOL
VAR_INPUT
	pAnalysis: POINTER TO FB_Analysis;
END_VAR
VAR
END_VAR

ValueMapping(pAnalysis);

//The BatchNShift 1Ch buffers input values with the configured buffer size and buffer mode.
fbM1_BatchNShift1Ch.Call(pAnalysis^.nContext);

//The Math Operation executes a mathematical operation on two or more different input channels and provides the result of the mathematical operation. The operator can be configured individually. Optional a boolean signal for Enable Execution can be selected, so that the algorithm is just active if the value of the selected signal is TRUE.
fbM2_MathOperation.fDataInCh2:= fbM1_BatchNShift1Ch.aOutputValues[2];
fbM2_MathOperation.Call(pAnalysis^.nContext);

//The Edge Counter 1Ch counts the amount of raised events. An event is raised when the signal of the input channel passes the configured edge at a specific threshold. Optional a boolean signal for Enable Execution can be selected, so that the algorithm is just active if the value of the selected signal is TRUE.
fbM3_EdgeCounter1Ch.fDataIn:= fbM2_MathOperation.fResult;
fbM3_EdgeCounter1Ch.Call(pAnalysis^.nContext);

//Networkoutput mapping
nTotalCount:= fbM3_EdgeCounter1Ch.nCount;


//Error Handling
IF fbM1_BatchNShift1Ch.bError THEN
	bError:= TRUE;
	ipTcResult:= fbM1_BatchNShift1Ch.ipTcResult;
ELSIF fbM2_MathOperation.bError THEN
	bError:= TRUE;
	ipTcResult:= fbM2_MathOperation.ipTcResult;
ELSIF fbM3_EdgeCounter1Ch.bError THEN
	bError:= TRUE;
	ipTcResult:= fbM3_EdgeCounter1Ch.ipTcResult;
ELSE
	bError:= FALSE;
	ipTcResult:= fbTcMsgSuccess;
END_IF
END_METHOD

METHOD Reset : BOOL
VAR
	bResult: BOOL := TRUE;
END_VAR
bResult:= bResult AND fbM1_BatchNShift1Ch.Reset();
bResult:= bResult AND fbM2_MathOperation.Reset();
bResult:= bResult AND fbM3_EdgeCounter1Ch.Reset();
Reset:= bResult;
END_METHOD

METHOD PRIVATE ValueMapping : BOOL
VAR_INPUT
	pAnalysis: POINTER TO FB_Analysis;
END_VAR
VAR
END_VAR

//Networkinput mapping
nOngoingCount:= pAnalysis^.ipVirtual_Input_Source.nV1_nUnitsProduced;

//Module fbM1_BatchNShift1Ch
fbM1_BatchNShift1Ch.nDataIn:= nOngoingCount;

//Module fbM2_MathOperation
fbM2_MathOperation.nDataInCh1:= nOngoingCount;

//Module fbM3_EdgeCounter1Ch
fbM3_EdgeCounter1Ch.tTimestamp:= pAnalysis^.ipVirtual_Input_Source.tTimestamp;
END_METHOD

END_FUNCTION_BLOCK

// ---- POUs/Analytics/Analysis/Networks/N01 OEEDashboard/N02 Products_Produced/Modules/FB_N2_M1_BatchNShift1Ch.TcPOU
//The BatchNShift 1Ch buffers input values with the configured buffer size and buffer mode.
FUNCTION_BLOCK FB_N2_M1_BatchNShift1Ch
VAR_INPUT
	nDataIn: ULINT; 
	bEnableExecution: BOOL := TRUE; 
	bReset: BOOL; 
	bReconfigure: BOOL := TRUE;
END_VAR
VAR_INPUT PERSISTENT
	eSampleMode: E_ALY_SampleMode; 
END_VAR
VAR_OUTPUT
	bError: BOOL;
	ipTcResult: I_TcMessage;
	bNewResult: BOOL;
	aOutputValues: ARRAY [0..2] OF LREAL;
END_VAR
VAR
	
	R_TRIG_Reconfigure: R_TRIG;
	
	fbALY_BatchNShift_1Ch: FB_ALY_BatchNShift_1Ch(nBufferSize:=3);
END_VAR
VAR PERSISTENT
	bConfigured: BOOL;
END_VAR

METHOD Call : BOOL
VAR_INPUT
	nCurrentContext: DWORD;
END_VAR
VAR
END_VAR
IF NOT bConfigured THEN
	bConfigured:= TRUE;

	eSampleMode:= E_ALY_SampleMode.Flow;

END_IF

R_TRIG_Reconfigure(CLK:= bReconfigure);
IF R_TRIG_Reconfigure.Q THEN
	fbALY_BatchNShift_1Ch.Configure(eSampleMode:= eSampleMode);

	bReconfigure:= FALSE;
END_IF

IF bReset THEN
	Reset();
END_IF

IF bEnableExecution THEN
	IF F_HasContext(nCurrentContext, nContext) THEN
		fbALY_BatchNShift_1Ch.SetChannelValue(Input:= nDataIn);

		fbALY_BatchNShift_1Ch.Call();

		bNewResult:= fbALY_BatchNShift_1Ch.bNewResult;

		fbALY_BatchNShift_1Ch.GetOutputArray(pArrayOut:= ADR(aOutputValues), nArrayOutSize:= SIZEOF(aOutputValues));

		bError:= fbALY_BatchNShift_1Ch.bError;
		ipTcResult:= fbALY_BatchNShift_1Ch.ipResultMessage;
	END_IF
ELSE
	bNewResult:= FALSE;
END_IF
END_METHOD

METHOD Reset : BOOL
VAR
END_VAR
Reset:= fbALY_BatchNShift_1Ch.Reset();

bNewResult:= fbALY_BatchNShift_1Ch.bNewResult;

fbALY_BatchNShift_1Ch.GetOutputArray(pArrayOut:= ADR(aOutputValues), nArrayOutSize:= SIZEOF(aOutputValues));

bError:= NOT Reset;
ipTcResult:= fbALY_BatchNShift_1Ch.ipResultMessage;
END_METHOD

PROPERTY nContext : DWORD
GET
nContext:= E_VirtualInput.eContext_V1_Virtual_Input_Source;
END_GET
END_PROPERTY

END_FUNCTION_BLOCK

// ---- POUs/Analytics/Analysis/Networks/N01 OEEDashboard/N02 Products_Produced/Modules/FB_N2_M2_MathOperation.TcPOU
//The Math Operation executes a mathematical operation on two or more different input channels and provides the result of the mathematical operation. The operator can be configured individually. Optional a boolean signal for Enable Execution can be selected, so that the algorithm is just active if the value of the selected signal is TRUE.
FUNCTION_BLOCK FB_N2_M2_MathOperation
VAR_INPUT
	nDataInCh1: ULINT; 
	fDataInCh2: LREAL; 
	bEnableExecution: BOOL := TRUE; 
	bReset: BOOL; 
	bReconfigure: BOOL := TRUE;
END_VAR
VAR_INPUT PERSISTENT
	eMathOperator: E_ALY_MathOperator; 
	bUseAbsValues: BOOL; 
END_VAR
VAR_OUTPUT
	bError: BOOL;
	ipTcResult: I_TcMessage;
	bNewResult: BOOL;
	fResult: LREAL;
END_VAR
VAR
	
	R_TRIG_Reconfigure: R_TRIG;
	
	fbALY_MathOperation: FB_ALY_MathOperation(nNumChannels:=2);
END_VAR
VAR PERSISTENT
	bConfigured: BOOL;
END_VAR

METHOD Call : BOOL
VAR_INPUT
	nCurrentContext: DWORD;
END_VAR
VAR
END_VAR
IF NOT bConfigured THEN
	bConfigured:= TRUE;

	eMathOperator:= E_ALY_MathOperator.Subtraction;
	bUseAbsValues:= FALSE;

END_IF

R_TRIG_Reconfigure(CLK:= bReconfigure);
IF R_TRIG_Reconfigure.Q THEN
	fbALY_MathOperation.Configure(eMathOperator:= eMathOperator, bUseAbsValues:= bUseAbsValues);

	bReconfigure:= FALSE;
END_IF

IF bReset THEN
	Reset();
END_IF

IF bEnableExecution THEN
	IF F_HasContext(nCurrentContext, nContext) THEN
		fbALY_MathOperation.SetChannelValue(nChannel:= 1, Input:= nDataInCh1);
		fbALY_MathOperation.SetChannelValue(nChannel:= 2, Input:= fDataInCh2);

		fbALY_MathOperation.Call();


		bNewResult:= fbALY_MathOperation.bNewResult;
		fResult:= fbALY_MathOperation.fResult;

		bError:= fbALY_MathOperation.bError;
		ipTcResult:= fbALY_MathOperation.ipResultMessage;
	END_IF
ELSE
	bNewResult:= FALSE;
END_IF
END_METHOD

METHOD Reset : BOOL
VAR
END_VAR
Reset:= fbALY_MathOperation.Reset();

bNewResult:= fbALY_MathOperation.bNewResult;
fResult:= fbALY_MathOperation.fResult;

bError:= NOT Reset;
ipTcResult:= fbALY_MathOperation.ipResultMessage;
END_METHOD

PROPERTY nContext : DWORD
GET
nContext:= E_VirtualInput.eContext_V1_Virtual_Input_Source;
END_GET
END_PROPERTY

END_FUNCTION_BLOCK

// ---- POUs/Analytics/Analysis/Networks/N01 OEEDashboard/N02 Products_Produced/Modules/FB_N2_M3_EdgeCounter1Ch.TcPOU
//The Edge Counter 1Ch counts the amount of raised events. An event is raised when the signal of the input channel passes the configured edge at a specific threshold. Optional a boolean signal for Enable Execution can be selected, so that the algorithm is just active if the value of the selected signal is TRUE.
FUNCTION_BLOCK FB_N2_M3_EdgeCounter1Ch
VAR_INPUT
	fDataIn: LREAL; 
	tTimestamp: ULINT; 
	bEnableExecution: BOOL := TRUE; 
	bReset: BOOL; 
	bReconfigure: BOOL := TRUE;
END_VAR
VAR_INPUT PERSISTENT
	stThresholdEdge: ST_ALY_Threshold; 
	fTolerance: LREAL; 
END_VAR
VAR_OUTPUT
	bError: BOOL;
	ipTcResult: I_TcMessage;
	bNewResult: BOOL;
	bEdge: BOOL;
	nCount: ULINT;
	fbTimeLastEvent: FB_ALY_DateTime;
END_VAR
VAR
	
	R_TRIG_Reconfigure: R_TRIG;
	
	fbALY_EdgeCounter_1Ch: FB_ALY_EdgeCounter_1Ch := ( bPersistent:= TRUE );
END_VAR
VAR PERSISTENT
	bConfigured: BOOL;
END_VAR

METHOD Call : BOOL
VAR_INPUT
	nCurrentContext: DWORD;
END_VAR
VAR
END_VAR
IF NOT bConfigured THEN
	bConfigured:= TRUE;

	fTolerance:= 0;

	stThresholdEdge.eComparisonOperator:= E_ALY_ComparisonOperator.GreaterThanOrEqualTo;
	stThresholdEdge.fThreshold:= 1;

	fbALY_EdgeCounter_1Ch.fTolerance:= fTolerance;
END_IF

R_TRIG_Reconfigure(CLK:= bReconfigure);
IF R_TRIG_Reconfigure.Q THEN
	fbALY_EdgeCounter_1Ch.ConfigureChannel(stThresholdEdge:= stThresholdEdge);

	fbALY_EdgeCounter_1Ch.Configure();

	bReconfigure:= FALSE;
END_IF

IF bReset THEN
	Reset();
END_IF

IF bEnableExecution THEN
	IF F_HasContext(nCurrentContext, nContext) THEN
		fbALY_EdgeCounter_1Ch.SetChannelValue(Input:= fDataIn);

		fbALY_EdgeCounter_1Ch.Call(tTimestamp:= tTimestamp);

		bNewResult:= fbALY_EdgeCounter_1Ch.bNewResult;
		bEdge:= fbALY_EdgeCounter_1Ch.bEdge;
		nCount:= fbALY_EdgeCounter_1Ch.nCount;
		fbTimeLastEvent:= fbALY_EdgeCounter_1Ch.fbTimeLastEvent;

		bError:= fbALY_EdgeCounter_1Ch.bError;
		ipTcResult:= fbALY_EdgeCounter_1Ch.ipResultMessage;
	END_IF
ELSE
	bNewResult:= FALSE;
END_IF
END_METHOD

METHOD Reset : BOOL
VAR
END_VAR
Reset:= fbALY_EdgeCounter_1Ch.Reset();

bNewResult:= fbALY_EdgeCounter_1Ch.bNewResult;
bEdge:= fbALY_EdgeCounter_1Ch.bEdge;
nCount:= fbALY_EdgeCounter_1Ch.nCount;
fbTimeLastEvent:= fbALY_EdgeCounter_1Ch.fbTimeLastEvent;

bError:= NOT Reset;
ipTcResult:= fbALY_EdgeCounter_1Ch.ipResultMessage;
END_METHOD

PROPERTY nContext : DWORD
GET
nContext:= E_VirtualInput.eContext_V1_Virtual_Input_Source;
END_GET
END_PROPERTY

END_FUNCTION_BLOCK

// ---- POUs/Analytics/Analysis/Networks/N01 OEEDashboard/N03 Products_Defective/FB_N3_Products_Defective.TcPOU
//Analytics Network "Products_Defective" with ID: 3
{attribute 'no_assign'}
FUNCTION_BLOCK FB_N3_Products_Defective
VAR_INPUT
	nOngoingCount: ULINT;
END_VAR
VAR_OUTPUT
	bError: BOOL;
	ipTcResult: I_TcMessage := fbTcMsgSuccess;
	nTotalCount: ULINT;
END_VAR
VAR
	fbTcMsgSuccess: FB_TcMessageSuccess;
	
	//Modules
	fbM1_BatchNShift1Ch: FB_N3_M1_BatchNShift1Ch;
	fbM2_MathOperation: FB_N3_M2_MathOperation;
	fbM3_EdgeCounter1Ch: FB_N3_M3_EdgeCounter1Ch;
END_VAR

METHOD Call : BOOL
VAR_INPUT
	pAnalysis: POINTER TO FB_Analysis;
END_VAR
VAR
END_VAR

ValueMapping(pAnalysis);

//The BatchNShift 1Ch buffers input values with the configured buffer size and buffer mode.
fbM1_BatchNShift1Ch.Call(pAnalysis^.nContext);

//The Math Operation executes a mathematical operation on two or more different input channels and provides the result of the mathematical operation. The operator can be configured individually. Optional a boolean signal for Enable Execution can be selected, so that the algorithm is just active if the value of the selected signal is TRUE.
fbM2_MathOperation.fDataInCh2:= fbM1_BatchNShift1Ch.aOutputValues[2];
fbM2_MathOperation.Call(pAnalysis^.nContext);

//The Edge Counter 1Ch counts the amount of raised events. An event is raised when the signal of the input channel passes the configured edge at a specific threshold. Optional a boolean signal for Enable Execution can be selected, so that the algorithm is just active if the value of the selected signal is TRUE.
fbM3_EdgeCounter1Ch.fDataIn:= fbM2_MathOperation.fResult;
fbM3_EdgeCounter1Ch.Call(pAnalysis^.nContext);

//Networkoutput mapping
nTotalCount:= fbM3_EdgeCounter1Ch.nCount;


//Error Handling
IF fbM1_BatchNShift1Ch.bError THEN
	bError:= TRUE;
	ipTcResult:= fbM1_BatchNShift1Ch.ipTcResult;
ELSIF fbM2_MathOperation.bError THEN
	bError:= TRUE;
	ipTcResult:= fbM2_MathOperation.ipTcResult;
ELSIF fbM3_EdgeCounter1Ch.bError THEN
	bError:= TRUE;
	ipTcResult:= fbM3_EdgeCounter1Ch.ipTcResult;
ELSE
	bError:= FALSE;
	ipTcResult:= fbTcMsgSuccess;
END_IF
END_METHOD

METHOD Reset : BOOL
VAR
	bResult: BOOL := TRUE;
END_VAR
bResult:= bResult AND fbM1_BatchNShift1Ch.Reset();
bResult:= bResult AND fbM2_MathOperation.Reset();
bResult:= bResult AND fbM3_EdgeCounter1Ch.Reset();
Reset:= bResult;
END_METHOD

METHOD PRIVATE ValueMapping : BOOL
VAR_INPUT
	pAnalysis: POINTER TO FB_Analysis;
END_VAR
VAR
END_VAR

//Networkinput mapping
nOngoingCount:= pAnalysis^.ipVirtual_Input_Source.nV1_nDefectiveUnits;

//Module fbM1_BatchNShift1Ch
fbM1_BatchNShift1Ch.nDataIn:= nOngoingCount;

//Module fbM2_MathOperation
fbM2_MathOperation.nDataInCh1:= nOngoingCount;

//Module fbM3_EdgeCounter1Ch
fbM3_EdgeCounter1Ch.tTimestamp:= pAnalysis^.ipVirtual_Input_Source.tTimestamp;
END_METHOD

END_FUNCTION_BLOCK

// ---- POUs/Analytics/Analysis/Networks/N01 OEEDashboard/N03 Products_Defective/Modules/FB_N3_M1_BatchNShift1Ch.TcPOU
//The BatchNShift 1Ch buffers input values with the configured buffer size and buffer mode.
FUNCTION_BLOCK FB_N3_M1_BatchNShift1Ch
VAR_INPUT
	nDataIn: ULINT; 
	bEnableExecution: BOOL := TRUE; 
	bReset: BOOL; 
	bReconfigure: BOOL := TRUE;
END_VAR
VAR_INPUT PERSISTENT
	eSampleMode: E_ALY_SampleMode; 
END_VAR
VAR_OUTPUT
	bError: BOOL;
	ipTcResult: I_TcMessage;
	bNewResult: BOOL;
	aOutputValues: ARRAY [0..2] OF LREAL;
END_VAR
VAR
	
	R_TRIG_Reconfigure: R_TRIG;
	
	fbALY_BatchNShift_1Ch: FB_ALY_BatchNShift_1Ch(nBufferSize:=3);
END_VAR
VAR PERSISTENT
	bConfigured: BOOL;
END_VAR

METHOD Call : BOOL
VAR_INPUT
	nCurrentContext: DWORD;
END_VAR
VAR
END_VAR
IF NOT bConfigured THEN
	bConfigured:= TRUE;

	eSampleMode:= E_ALY_SampleMode.Flow;

END_IF

R_TRIG_Reconfigure(CLK:= bReconfigure);
IF R_TRIG_Reconfigure.Q THEN
	fbALY_BatchNShift_1Ch.Configure(eSampleMode:= eSampleMode);

	bReconfigure:= FALSE;
END_IF

IF bReset THEN
	Reset();
END_IF

IF bEnableExecution THEN
	IF F_HasContext(nCurrentContext, nContext) THEN
		fbALY_BatchNShift_1Ch.SetChannelValue(Input:= nDataIn);

		fbALY_BatchNShift_1Ch.Call();

		bNewResult:= fbALY_BatchNShift_1Ch.bNewResult;

		fbALY_BatchNShift_1Ch.GetOutputArray(pArrayOut:= ADR(aOutputValues), nArrayOutSize:= SIZEOF(aOutputValues));

		bError:= fbALY_BatchNShift_1Ch.bError;
		ipTcResult:= fbALY_BatchNShift_1Ch.ipResultMessage;
	END_IF
ELSE
	bNewResult:= FALSE;
END_IF
END_METHOD

METHOD Reset : BOOL
VAR
END_VAR
Reset:= fbALY_BatchNShift_1Ch.Reset();

bNewResult:= fbALY_BatchNShift_1Ch.bNewResult;

fbALY_BatchNShift_1Ch.GetOutputArray(pArrayOut:= ADR(aOutputValues), nArrayOutSize:= SIZEOF(aOutputValues));

bError:= NOT Reset;
ipTcResult:= fbALY_BatchNShift_1Ch.ipResultMessage;
END_METHOD

PROPERTY nContext : DWORD
GET
nContext:= E_VirtualInput.eContext_V1_Virtual_Input_Source;
END_GET
END_PROPERTY

END_FUNCTION_BLOCK

// ---- POUs/Analytics/Analysis/Networks/N01 OEEDashboard/N03 Products_Defective/Modules/FB_N3_M2_MathOperation.TcPOU
//The Math Operation executes a mathematical operation on two or more different input channels and provides the result of the mathematical operation. The operator can be configured individually. Optional a boolean signal for Enable Execution can be selected, so that the algorithm is just active if the value of the selected signal is TRUE.
FUNCTION_BLOCK FB_N3_M2_MathOperation
VAR_INPUT
	nDataInCh1: ULINT; 
	fDataInCh2: LREAL; 
	bEnableExecution: BOOL := TRUE; 
	bReset: BOOL; 
	bReconfigure: BOOL := TRUE;
END_VAR
VAR_INPUT PERSISTENT
	eMathOperator: E_ALY_MathOperator; 
	bUseAbsValues: BOOL; 
END_VAR
VAR_OUTPUT
	bError: BOOL;
	ipTcResult: I_TcMessage;
	bNewResult: BOOL;
	fResult: LREAL;
END_VAR
VAR
	
	R_TRIG_Reconfigure: R_TRIG;
	
	fbALY_MathOperation: FB_ALY_MathOperation(nNumChannels:=2);
END_VAR
VAR PERSISTENT
	bConfigured: BOOL;
END_VAR

METHOD Call : BOOL
VAR_INPUT
	nCurrentContext: DWORD;
END_VAR
VAR
END_VAR
IF NOT bConfigured THEN
	bConfigured:= TRUE;

	eMathOperator:= E_ALY_MathOperator.Subtraction;
	bUseAbsValues:= FALSE;

END_IF

R_TRIG_Reconfigure(CLK:= bReconfigure);
IF R_TRIG_Reconfigure.Q THEN
	fbALY_MathOperation.Configure(eMathOperator:= eMathOperator, bUseAbsValues:= bUseAbsValues);

	bReconfigure:= FALSE;
END_IF

IF bReset THEN
	Reset();
END_IF

IF bEnableExecution THEN
	IF F_HasContext(nCurrentContext, nContext) THEN
		fbALY_MathOperation.SetChannelValue(nChannel:= 1, Input:= nDataInCh1);
		fbALY_MathOperation.SetChannelValue(nChannel:= 2, Input:= fDataInCh2);

		fbALY_MathOperation.Call();


		bNewResult:= fbALY_MathOperation.bNewResult;
		fResult:= fbALY_MathOperation.fResult;

		bError:= fbALY_MathOperation.bError;
		ipTcResult:= fbALY_MathOperation.ipResultMessage;
	END_IF
ELSE
	bNewResult:= FALSE;
END_IF
END_METHOD

METHOD Reset : BOOL
VAR
END_VAR
Reset:= fbALY_MathOperation.Reset();

bNewResult:= fbALY_MathOperation.bNewResult;
fResult:= fbALY_MathOperation.fResult;

bError:= NOT Reset;
ipTcResult:= fbALY_MathOperation.ipResultMessage;
END_METHOD

PROPERTY nContext : DWORD
GET
nContext:= E_VirtualInput.eContext_V1_Virtual_Input_Source;
END_GET
END_PROPERTY

END_FUNCTION_BLOCK

// ---- POUs/Analytics/Analysis/Networks/N01 OEEDashboard/N03 Products_Defective/Modules/FB_N3_M3_EdgeCounter1Ch.TcPOU
//The Edge Counter 1Ch counts the amount of raised events. An event is raised when the signal of the input channel passes the configured edge at a specific threshold. Optional a boolean signal for Enable Execution can be selected, so that the algorithm is just active if the value of the selected signal is TRUE.
FUNCTION_BLOCK FB_N3_M3_EdgeCounter1Ch
VAR_INPUT
	fDataIn: LREAL; 
	tTimestamp: ULINT; 
	bEnableExecution: BOOL := TRUE; 
	bReset: BOOL; 
	bReconfigure: BOOL := TRUE;
END_VAR
VAR_INPUT PERSISTENT
	stThresholdEdge: ST_ALY_Threshold; 
	fTolerance: LREAL; 
END_VAR
VAR_OUTPUT
	bError: BOOL;
	ipTcResult: I_TcMessage;
	bNewResult: BOOL;
	bEdge: BOOL;
	nCount: ULINT;
	fbTimeLastEvent: FB_ALY_DateTime;
END_VAR
VAR
	
	R_TRIG_Reconfigure: R_TRIG;
	
	fbALY_EdgeCounter_1Ch: FB_ALY_EdgeCounter_1Ch := ( bPersistent:= TRUE );
END_VAR
VAR PERSISTENT
	bConfigured: BOOL;
END_VAR

METHOD Call : BOOL
VAR_INPUT
	nCurrentContext: DWORD;
END_VAR
VAR
END_VAR
IF NOT bConfigured THEN
	bConfigured:= TRUE;

	fTolerance:= 0;

	stThresholdEdge.eComparisonOperator:= E_ALY_ComparisonOperator.GreaterThanOrEqualTo;
	stThresholdEdge.fThreshold:= 1;

	fbALY_EdgeCounter_1Ch.fTolerance:= fTolerance;
END_IF

R_TRIG_Reconfigure(CLK:= bReconfigure);
IF R_TRIG_Reconfigure.Q THEN
	fbALY_EdgeCounter_1Ch.ConfigureChannel(stThresholdEdge:= stThresholdEdge);

	fbALY_EdgeCounter_1Ch.Configure();

	bReconfigure:= FALSE;
END_IF

IF bReset THEN
	Reset();
END_IF

IF bEnableExecution THEN
	IF F_HasContext(nCurrentContext, nContext) THEN
		fbALY_EdgeCounter_1Ch.SetChannelValue(Input:= fDataIn);

		fbALY_EdgeCounter_1Ch.Call(tTimestamp:= tTimestamp);

		bNewResult:= fbALY_EdgeCounter_1Ch.bNewResult;
		bEdge:= fbALY_EdgeCounter_1Ch.bEdge;
		nCount:= fbALY_EdgeCounter_1Ch.nCount;
		fbTimeLastEvent:= fbALY_EdgeCounter_1Ch.fbTimeLastEvent;

		bError:= fbALY_EdgeCounter_1Ch.bError;
		ipTcResult:= fbALY_EdgeCounter_1Ch.ipResultMessage;
	END_IF
ELSE
	bNewResult:= FALSE;
END_IF
END_METHOD

METHOD Reset : BOOL
VAR
END_VAR
Reset:= fbALY_EdgeCounter_1Ch.Reset();

bNewResult:= fbALY_EdgeCounter_1Ch.bNewResult;
bEdge:= fbALY_EdgeCounter_1Ch.bEdge;
nCount:= fbALY_EdgeCounter_1Ch.nCount;
fbTimeLastEvent:= fbALY_EdgeCounter_1Ch.fbTimeLastEvent;

bError:= NOT Reset;
ipTcResult:= fbALY_EdgeCounter_1Ch.ipResultMessage;
END_METHOD

PROPERTY nContext : DWORD
GET
nContext:= E_VirtualInput.eContext_V1_Virtual_Input_Source;
END_GET
END_PROPERTY

END_FUNCTION_BLOCK

// ---- POUs/MAIN.TcPOU
PROGRAM MAIN
VAR
END_VAR

END_PROGRAM

// ---- POUs/Analytics/Sources/T1_InputSource/FB_T1_InputSource.TcPOU
FUNCTION_BLOCK FB_T1_InputSource IMPLEMENTS I_InputSource
VAR
	_eDataState: E_DataSourceState;
	
	_nMaxOversamplingFactor: UDINT := 1;
	
	_nElements: UDINT;
	_nCurrentElement: UDINT;
	_nDataHandle: ULINT;
	
	_nClientListHash: LWORD;
	_nCurrentClientHash: LWORD;
	
	_stInputs: ST_T1_Inputs;
	
	fbIotSymbol_GVL_Components_fbMachine_stAnalytics_nState: FB_ALY_IotSymbol_UINT := (stConfig:= (sSymbolName:= 'GVL_Components.fbMachine.stAnalytics.nState'));
	fbIotSymbol_GVL_Components_fbMachine_stAnalytics_nUnitsProduced: FB_ALY_IotSymbol_ULINT := (stConfig:= (sSymbolName:= 'GVL_Components.fbMachine.stAnalytics.nUnitsProduced'));
	fbIotSymbol_GVL_Components_fbMachine_stAnalytics_nDefectiveUnits: FB_ALY_IotSymbol_ULINT := (stConfig:= (sSymbolName:= 'GVL_Components.fbMachine.stAnalytics.nDefectiveUnits'));
	fbIotSymbol_GVL_Components_fbMachine_stAnalytics_tMlCalculation: FB_ALY_IotSymbol_UDINT := (stConfig:= (sSymbolName:= 'GVL_Components.fbMachine.stAnalytics.tMlCalculation'));
	
	//Target T1 = Broker:"localhost" Topic:"DefaultMainTopic/PlcStream1"
	fbStreamHelper: FB_ALY_StreamHelper;
	bConfigured: BOOL := FALSE;
	
	fbTON_DataTimeout: TON;
END_VAR
VAR_STAT
	_nClientIndex: INT;
END_VAR

METHOD AddClient : BOOL
VAR_OUTPUT
	nClientID: LWORD;
END_VAR
VAR
END_VAR
nClientID:= TO_LWORD(EXPT(2,_nClientIndex));
_nClientIndex:= _nClientIndex + 1;

_nClientListHash:= _nClientListHash + nClientID;
END_METHOD

PROPERTY bReadNewData : BOOL
GET
bReadNewData:= _nElements = 0 OR _nCurrentClientHash >= _nClientListHash;
END_GET
END_PROPERTY

METHOD Call : BOOL
VAR
	stConfig: ST_ALY_StreamHelper_Config;
END_VAR
IF NOT fbStreamHelper.bConfigured THEN
	stConfig.nObjectID:= 16#01010110;
	stConfig.nNumInputBuffer:= 20;
	fbStreamHelper.Configure(stConfig);
END_IF

IF NOT bConfigured THEN
	//GVL_Components.fbMachine.stAnalytics.nState
	fbStreamHelper.AddIotSymbol(fbIotSymbol_GVL_Components_fbMachine_stAnalytics_nState);
	//GVL_Components.fbMachine.stAnalytics.nUnitsProduced
	fbStreamHelper.AddIotSymbol(fbIotSymbol_GVL_Components_fbMachine_stAnalytics_nUnitsProduced);
	//GVL_Components.fbMachine.stAnalytics.nDefectiveUnits
	fbStreamHelper.AddIotSymbol(fbIotSymbol_GVL_Components_fbMachine_stAnalytics_nDefectiveUnits);
	//GVL_Components.fbMachine.stAnalytics.tMlCalculation
	fbStreamHelper.AddIotSymbol(fbIotSymbol_GVL_Components_fbMachine_stAnalytics_tMlCalculation);

	bConfigured:= TRUE;
END_IF

fbStreamHelper.Call();
IF fbStreamHelper.bError THEN
	_eDataState:= E_DataSourceState.eError;
ELSIF NOT fbStreamHelper.bConnected THEN
	_eDataState:= E_DataSourceState.eNotConnected;
ELSE
	_nElements:= fbStreamHelper.nNumElements;
	IF _nElements > 0 THEN
		_eDataState:= E_DataSourceState.eReceiveData;
	END_IF

	fbTON_DataTimeout(IN:= _nElements = 0, PT:= T#5S);
	IF fbTON_DataTimeout.Q THEN
		_eDataState:= E_DataSourceState.eWaitForData;
	END_IF
END_IF

IF _nElements > 0 THEN
	_nDataHandle:= _nDataHandle + 1;
	_nCurrentClientHash:= 0;
END_IF

_nCurrentElement:= 0;
END_METHOD

METHOD ClientDone : BOOL
VAR_INPUT
	nClientID: LWORD;
END_VAR
VAR
END_VAR
_nCurrentClientHash:=  _nCurrentClientHash + nClientID;
END_METHOD

PROPERTY eDataState : E_DataSourceState
GET
eDataState:= _eDataState;
END_GET
END_PROPERTY

METHOD GetData : BOOL
VAR_INPUT
	nElement: UDINT;
	pInputs: PVOID;
	nInputsSize: UDINT;
END_VAR
VAR_OUTPUT
	nTimestamp: ULINT;
	nContext: DWORD;
END_VAR
VAR
	_nElement: UDINT;
	_pInputs: PVOID;
	_nInputsSize: UDINT;
END_VAR
Analytics.fbT1_IecCriticalSection.Enter();

_nElement:= nElement;
_pInputs:= pInputs;
_nInputsSize:= nInputsSize;

nContext:= 0;
IF nElements > 0 THEN
	IF _nElement <= nElements THEN

		IF _nCurrentElement <> _nElement THEN

			//Set local raw inputs
			_stInputs.nGVL_Components_fbMachine_stAnalytics_nState:= fbIotSymbol_GVL_Components_fbMachine_stAnalytics_nState.GetValue(_nElement);
			_stInputs.nGVL_Components_fbMachine_stAnalytics_nUnitsProduced:= fbIotSymbol_GVL_Components_fbMachine_stAnalytics_nUnitsProduced.GetValue(_nElement);
			_stInputs.nGVL_Components_fbMachine_stAnalytics_nDefectiveUnits:= fbIotSymbol_GVL_Components_fbMachine_stAnalytics_nDefectiveUnits.GetValue(_nElement);
			_stInputs.nGVL_Components_fbMachine_stAnalytics_tMlCalculation:= fbIotSymbol_GVL_Components_fbMachine_stAnalytics_tMlCalculation.GetValue(_nElement);

			nContext:= E_DataSourceContext.eContext_1000;
			_nCurrentElement:= _nElement;
		END_IF

		//Set output values
		IF _pInputs > 0 THEN
			MEMCPY(_pInputs, ADR(_stInputs), _nInputsSize);
			nTimestamp:= fbStreamHelper.GetTimestampElement(_nElement);
		END_IF
	END_IF
	GetData:= TRUE;
ELSE
	GetData:= FALSE;
END_IF

Analytics.fbT1_IecCriticalSection.Leave();
END_METHOD

PROPERTY nDataHandle : ULINT
GET
nDataHandle:= _nDataHandle;
END_GET
END_PROPERTY

PROPERTY nElements : UDINT
GET
nElements:= _nElements;
END_GET
END_PROPERTY

METHOD NewDataAvailable : BOOL
VAR_INPUT
	nLastDataHandle: ULINT;
END_VAR
VAR
END_VAR
NewDataAvailable:= _nElements > 0 AND _nDataHandle <> nLastDataHandle;
END_METHOD

PROPERTY nMaxOversamplingFactor : UDINT
GET
nMaxOversamplingFactor:= _nMaxOversamplingFactor;
END_GET
END_PROPERTY

END_FUNCTION_BLOCK

// ---- POUs/Analytics/[Helper]/FB_DataBuffer.TcPOU
FUNCTION_BLOCK FB_DataBuffer
VAR_OUTPUT
	nElements: UDINT;
END_VAR
VAR
	_nDataSize: UDINT;
	
	_pWriteBuffer: POINTER TO BYTE;
	_pWriteBufferTime: POINTER TO ARRAY [1..cEntryCount] OF ULINT;
	_pReadBuffer: POINTER TO BYTE;
	_pReadBufferTime: POINTER TO ARRAY [1..cEntryCount] OF ULINT;
	
	_pBuffer1: POINTER TO BYTE;
	_aBufferTime1: ARRAY [1..cEntryCount] OF ULINT;
	_pBuffer2: POINTER TO BYTE;
	_aBufferTime2: ARRAY [1..cEntryCount] OF ULINT;
	
	_nBufferIdx: INT := 1;
	
	_nBufferEntry_Add: UDINT;
	
	_bLock: BOOL;
	
END_VAR
VAR CONSTANT
	cEntryCount: UDINT := 25;
END_VAR

METHOD FB_init : BOOL
VAR_INPUT
	bInitRetains: BOOL; // if TRUE, the retain variables are initialized (warm start / cold start)
	bInCopyCode: BOOL; // if TRUE, the instance afterwards gets moved into the copy code (online change)
	nDataSize: UDINT;
END_VAR
VAR
END_VAR
IF NOT bInCopyCode THEN
	_nDataSize:= nDataSize;
	_Init();
END_IF
END_METHOD

METHOD FB_exit : BOOL
VAR_INPUT
	bInCopyCode: BOOL; // if TRUE, the exit method is called for exiting an instance that is copied afterwards (online change).
END_VAR
VAR
END_VAR
IF _pBuffer1 <> 0 THEN
	__DELETE(_pBuffer1);
END_IF

IF _pBuffer2 <> 0 THEN
	__DELETE(_pBuffer2);
END_IF

_pWriteBuffer:= 0;
_pWriteBufferTime:= 0;
_pReadBuffer:= 0;
_pReadBufferTime:= 0;

_nBufferIdx:= 0;
_nBufferEntry_Add:= 0;
END_METHOD

METHOD PRIVATE _Init : BOOL
VAR
END_VAR
IF _pBuffer1 <> 0 THEN
	__DELETE(_pBuffer1);
END_IF

IF _pBuffer2 <> 0 THEN
	__DELETE(_pBuffer2);
END_IF

_pBuffer1 := __NEW(BYTE, (_nDataSize * cEntryCount));
_pBuffer2 := __NEW(BYTE, (_nDataSize * cEntryCount));

_nBufferIdx:= 0;

Call();
END_METHOD

METHOD Call : BOOL
VAR
END_VAR
nElements:= 0;

IF TestAndSet(_bLock) THEN

